// TwinCAT 3 PLC project PLC
// ProgramVersion: 3.1.4024.0
// libraries:
//   Tc2_Standard, * (Beckhoff Automation GmbH)
//   Tc2_System, * (Beckhoff Automation GmbH)
//   Tc3_Module, * (Beckhoff Automation GmbH)
// project tree:
//   / PlcTask.TcTTO
//   POUs/Alarm/ GVL_Alarm.TcGVL
//   POUs/EL3453/ FB_EL3453.TcPOU, stEL3453.TcDUT, stEL3453_ch.TcDUT, stEL3453_tot.TcDUT
//   POUs/Example/ GVL_HMI.TcGVL, GVL_IO.TcGVL, GVL_Safety.TcGVL, GVL_System.TcGVL, PRG_CircuitBreakerExample.TcPOU, PRG_ContactorExample.TcPOU, PRG_DisconnectorExample.TcPOU, PRG_Simulation.TcPOU
//   POUs/HVCP3/ GVL_HVCP3.TcGVL, PRG_HVCP3.TcPOU, PRG_HVCP3_14CB1.TcPOU, PRG_HVCP3_16CB1.TcPOU, PRG_HVCP3_18CB1.TcPOU, PRG_HVCP3_20CB1.TcPOU, PRG_HVCP3_22CB1.TcPOU, PRG_HVCP3_24CB1.TcPOU, PRG_HVCP3_26CB1.TcPOU, PRG_HVCP3_28CB1.TcPOU, PRG_HVCP3_30CB1.TcPOU, PRG_HVCP3_32CB1.TcPOU, PRG_HVCP3_34CB1.TcPOU, PRG_HVCP3_36CB1.TcPOU, PRG_HVCP3_38CB1.TcPOU, PRG_HVCP3_40CB1.TcPOU, PRG_HVCP3_42CB1.TcPOU, PRG_HVCP3_44CB1.TcPOU, PRG_HVCP3_46CB1.TcPOU, PRG_HVCP3_48CB1.TcPOU, PRG_HVCP3_50CB1.TcPOU, PRG_HVCP3_52CB1.TcPOU, PRG_HVCP3_54CB1.TcPOU, PRG_HVCP3_56CB1.TcPOU, PRG_HVCP3_10CB1.TcPOU, PRG_HVCP3_12CB1.TcPOU
//   POUs/HVCP5/ GVL_HVCP5.TcGVL, PRG_HVCP5.TcPOU, PRG_HVCP5_12CB1.TcPOU, PRG_HVCP5_14CB1.TcPOU, PRG_HVCP5_16CB1.TcPOU, PRG_HVCP5_18CB1.TcPOU, PRG_HVCP5_20CB1.TcPOU, PRG_HVCP5_22CB1.TcPOU, PRG_HVCP5_24CB1.TcPOU, PRG_HVCP5_26CB1.TcPOU, PRG_HVCP5_28CB1.TcPOU, PRG_HVCP5_30CB1.TcPOU, PRG_HVCP5_32CB1.TcPOU, PRG_HVCP5_34CB1.TcPOU, PRG_HVCP5_36CB1.TcPOU, PRG_HVCP5_38CB1.TcPOU, PRG_HVCP5_10CB1.TcPOU
//   POUs/LVCP1/ GVL_LVCP1.TcGVL, PRG_LVCP1_Colors.TcPOU, PRG_LVCP1_CompensationCalculate.TcPOU, PRG_LVCP1_Group1.TcPOU, PRG_LVCP1.TcPOU, PRG_LVCP1_Group2.TcPOU, PRG_LVCP1_Group3.TcPOU, PRG_LVCP1_Group4.TcPOU, PRG_LVCP1_Group5.TcPOU, PRG_LVCP1_Group10.TcPOU, PRG_LVCP1_Group9.TcPOU, PRG_LVCP1_Group8.TcPOU, PRG_LVCP1_Group7.TcPOU, PRG_LVCP1_Group6.TcPOU, PRG_LVCP1_MainDisconnector.TcPOU, PRG_LVCP1_PowerMeasurement.TcPOU
//   POUs/LVCP2/ GVL_LVCP2.TcGVL, PRG_LVCP2_Colors.TcPOU, PRG_LVCP2_PowerMeasurement.TcPOU, PRG_LVCP2.TcPOU, PRG_LVCP2_CompensationCalculate.TcPOU, PRG_LVCP2_Group10.TcPOU, PRG_LVCP2_Group1.TcPOU, PRG_LVCP2_Group2.TcPOU, PRG_LVCP2_Group3.TcPOU, PRG_LVCP2_Group4.TcPOU, PRG_LVCP2_Group5.TcPOU, PRG_LVCP2_Group6.TcPOU, PRG_LVCP2_Group7.TcPOU, PRG_LVCP2_Group8.TcPOU, PRG_LVCP2_Group9.TcPOU, PRG_LVCP2_MainDisconnector.TcPOU
//   POUs/LVCP5/ GVL_LVCP5.TcGVL, PRG_LVCP5_Colors.TcPOU, PRG_LVCP5_PowerMeasurement.TcPOU, PRG_LVCP5_CompensationCalculate.TcPOU, PRG_LVCP5_Group7.TcPOU, PRG_LVCP5_Group6.TcPOU, PRG_LVCP5_Group5.TcPOU, PRG_LVCP5_Group4.TcPOU, PRG_LVCP5_Group3.TcPOU, PRG_LVCP5_Group2.TcPOU, PRG_LVCP5_Group1.TcPOU, PRG_LVCP5.TcPOU, PRG_LVCP5_MainCircuitBreaker.TcPOU
//   POUs/ MAIN.TcPOU
//   _ES/11_Disconnector/Enum/ E_DisconnectorControlMode.TcTLEO, E_DisconnectorFault.TcTLEO, E_DisconnectorPosition.TcTLEO, E_DisconnectorStatus.TcTLEO
//   _ES/11_Disconnector/ FB_DisconnectorControl.TcPOU
//   _ES/11_Disconnector/Structure/ ST_DisconnectorCommand.TcDUT, ST_DisconnectorConfig.TcDUT, ST_DisconnectorHMI.TcDUT, ST_DisconnectorIO.TcDUT, ST_DisconnectorOperationRecord.TcDUT, ST_DisconnectorStatistics.TcDUT, ST_DisconnectorStatus.TcDUT
//   _ES/12_Contactor/Enum/ E_ContactorControlMode.TcTLEO, E_ContactorFault.TcTLEO, E_ContactorPosition.TcTLEO, E_ContactorStatus.TcTLEO
//   _ES/12_Contactor/ FB_ContactorControl.TcPOU
//   _ES/12_Contactor/Structure/ ST_ContactorCommand.TcDUT, ST_ContactorConfig.TcDUT, ST_ContactorHMI.TcDUT, ST_ContactorIO.TcDUT, ST_ContactorOperationRecord.TcDUT, ST_ContactorStatistics.TcDUT, ST_ContactorStatus.TcDUT
//   _ES/13_CircuitBreaker/Enum/ E_CircuitBreakerControlMode.TcTLEO, E_CircuitBreakerFault.TcTLEO, E_CircuitBreakerPosition.TcTLEO, E_CircuitBreakerStatus.TcTLEO
//   _ES/13_CircuitBreaker/ FB_CircuitBreaker.TcPOU
//   _ES/13_CircuitBreaker/Structure/ ST_CircuitBreakerCommand.TcDUT, ST_CircuitBreakerConfig.TcDUT, ST_CircuitBreakerHMI.TcDUT, ST_CircuitBreakerIO.TcDUT, ST_CircuitBreakerOperationRecord.TcDUT, ST_CircuitBreakerStatistics.TcDUT, ST_CircuitBreakerStatus.TcDUT
//   _ES/14_CompensationGroup/Enum/ E_CompensationError.TcTLEO
//   _ES/14_CompensationGroup/ FB_CompensationCalculator.TcPOU, GVL_CompensationGroup.TcGVL
//   _ES/14_CompensationGroup/Structure/ ST_CompensationConfigInfo.TcDUT, ST_CompensationDiagnostic.TcDUT, ST_CompensationGroup.TcDUT, ST_CompensationGroupDetails.TcDUT, ST_CompensationHMI.TcDUT, ST_CompensationSummary.TcDUT
//   _ES/xx_Line/Enum/ E_LineColors.TcDUT
//   _ES/xx_Line/Structure/ ST_CapacitorSchemaColorBase.TcDUT, ST_CapacitorSchemaColorWithContactor.TcDUT, ST_CapacitorSchemaColorWithDisconnector.TcDUT
// real-time tasks:
//   TASK PlcTask: cycle T#10ms, priority 20, ADS port 350
// I/O:
//   DEVICE Device 1 (EtherCAT) (disabled), AmsNetId 192.168.35.154.2.1
//     +EP6-11CP1 (EK1100) [EK1100 EtherCAT Coupler (2A E-Bus)]
//       +EP6-11DI1 (EL1809) [EL1809 16Ch. Dig. Input 24V, 3ms]
//       +EP6-11DI2 (EL1809) [EL1809 16Ch. Dig. Input 24V, 3ms]
//       +EP6-11DQ1 (EL2809-0015) [EL2809-0015 16Ch. Dig. Output 24V DC, 0.35A, not short-circuit proof]
//       +EP6-11SDI1 (EL1918) [EL1918, 8Ch. Safety Input 24V, TwinSAFE]
//         modules: Module 1 (FSOE), Module 2 (FSLOGIC)
//       +EP6-11SDQ1 (EL2904) [EL2904, 4 Ch. Safety Output 24V, 0.5A, TwinSAFE]
//         modules: Module 1 (FSOES), Module 2 (DO)
//       +EP6-11AI1 (EL3453) [EL3453 3Ch. Power Measuring]
//       Term 8 (EL9010) [EL9010 End Terminal]
//     +EP7-11CP1 (EK1100) [EK1100 EtherCAT Coupler (2A E-Bus)]
//       +EP7-11DI1 (EL1809) [EL1809 16Ch. Dig. Input 24V, 3ms]
//       +EP7-11DI2 (EL1809) [EL1809 16Ch. Dig. Input 24V, 3ms]
//       +EP7-11DQ1 (EL2809-0015) [EL2809-0015 16Ch. Dig. Output 24V DC, 0.35A, not short-circuit proof]
//       +EP7-11SDI1 (EL1918) [EL1918, 8Ch. Safety Input 24V, TwinSAFE]
//         modules: Module 1 (FSOE), Module 2 (FSLOGIC)
//       +EP7-11SDQ1 (EL2904) [EL2904, 4 Ch. Safety Output 24V, 0.5A, TwinSAFE]
//         modules: Module 1 (FSOES), Module 2 (DO)
//       +EP7-11AI1 (EL3453) [EL3453 3Ch. Power Measuring]
//       Term 16 (EL9010) [EL9010 End Terminal]
//     +EP8-11CP1 (EK1100) [EK1100 EtherCAT Coupler (2A E-Bus)]
//       +EP8-11DI1 (EL1809) [EL1809 16Ch. Dig. Input 24V, 3ms]
//       +EP8-11DI2 (EL1809) [EL1809 16Ch. Dig. Input 24V, 3ms]
//       +EP8-11DQ1 (EL2809-0015) [EL2809-0015 16Ch. Dig. Output 24V DC, 0.35A, not short-circuit proof]
//       +EP8-11SDI1 (EL1918) [EL1918, 8Ch. Safety Input 24V, TwinSAFE]
//         modules: Module 1 (FSOE), Module 2 (FSLOGIC)
//       +EP8-11SDQ1 (EL2904) [EL2904, 4 Ch. Safety Output 24V, 0.5A, TwinSAFE]
//         modules: Module 1 (FSOES), Module 2 (DO)
//       +EP8-11AI1 (EL3453) [EL3453 3Ch. Power Measuring]
//       Term 24 (EL9010) [EL9010 End Terminal]
//     +EP9-5CP5 (EK1100) [EK1100 EtherCAT Coupler (2A E-Bus)]
//       +EP9-5DI1 (EL1809) [EL1809 16Ch. Dig. Input 24V, 3ms]
//       +EP9-5DI2 (EL1809) [EL1809 16Ch. Dig. Input 24V, 3ms]
//       +EP9-5DI3 (EL1809) [EL1809 16Ch. Dig. Input 24V, 3ms]
//       +EP9-5DI4 (EL1809) [EL1809 16Ch. Dig. Input 24V, 3ms]
//       +EP9-5DI5 (EL1809) [EL1809 16Ch. Dig. Input 24V, 3ms]
//       +EP9-5DQ1 (EL2809) [EL2809 16Ch. Dig. Output 24V, 0.5A]
//       +EP9-5DQ2 (EL2809) [EL2809 16Ch. Dig. Output 24V, 0.5A]
//       +EP9-5DQ3 (EL2809) [EL2809 16Ch. Dig. Output 24V, 0.5A]
//       +EP9-6SDI1 (EL1918) [EL1918, 8Ch. Safety Input 24V, TwinSAFE]
//         modules: Module 1 (FSOE), Module 2 (FSLOGIC)
//       +EP9-6SDQ1 (EL2904) [EL2904, 4 Ch. Safety Output 24V, 0.5A, TwinSAFE]
//         modules: Module 1 (FSOES), Module 2 (DO)
//       +EP9-6AI1 (EL3453) [EL3453 3Ch. Power Measuring]
//     +EP10-5CP5 (EK1100) [EK1100 EtherCAT Coupler (2A E-Bus)]
//       +EP10-5DI1 (EL1809) [EL1809 16Ch. Dig. Input 24V, 3ms]
//       +EP10-5DI2 (EL1809) [EL1809 16Ch. Dig. Input 24V, 3ms]
//       +EP10-5DI3 (EL1809) [EL1809 16Ch. Dig. Input 24V, 3ms]
//       +EP10-5DI4 (EL1809) [EL1809 16Ch. Dig. Input 24V, 3ms]
//       +EP10-5DQ1 (EL2809) [EL2809 16Ch. Dig. Output 24V, 0.5A]
//       +EP10-5DQ2 (EL2809) [EL2809 16Ch. Dig. Output 24V, 0.5A]
//       +EP10-6SDI1 (EL1918) [EL1918, 8Ch. Safety Input 24V, TwinSAFE]
//         modules: Module 1 (FSOE), Module 2 (FSLOGIC)
//       +EP10-6SDQ1 (EL2904) [EL2904, 4 Ch. Safety Output 24V, 0.5A, TwinSAFE]
//         modules: Module 1 (FSOES), Module 2 (DO)
//       +EP10-6AI1 (EL3453) [EL3453 3Ch. Power Measuring]
// variable links:
//   PLC/PLC Instance <-> Device 1 (EtherCAT)/+EP10-5CP5 (EK1100)/+EP10-5DI1 (EL1809)
//     PlcTask Inputs/GVL_Alarm.EP10_3X2_24VDC_OK <-> Channel 1/Input
//     PlcTask Inputs/GVL_Alarm.EP10_UPS_24VDC_OK <-> Channel 2/Input
//     PlcTask Inputs/PRG_HVCP5_10CB1.stDisconnectorIO.bEarthSwitchOff <-> Channel 7/Input
//     PlcTask Inputs/PRG_HVCP5_10CB1.stDisconnectorIO.bEarthSwitchOn <-> Channel 6/Input
//     PlcTask Inputs/PRG_HVCP5_10CB1.stDisconnectorIO.bLimitOff <-> Channel 4/Input
//     PlcTask Inputs/PRG_HVCP5_12CB1.stDisconnectorIO.bLimitOff <-> Channel 9/Input
//     PlcTask Inputs/PRG_HVCP5_14CB1.stDisconnectorIO.bLimitOff <-> Channel 12/Input
//     PlcTask Inputs/PRG_HVCP5_16CB1.stDisconnectorIO.bLimitOff <-> Channel 15/Input
//     PlcTask Inputs/PRG_HVCP5_10CB1.stDisconnectorIO.bLimitOn <-> Channel 3/Input
//     PlcTask Inputs/PRG_HVCP5_12CB1.stDisconnectorIO.bLimitOn <-> Channel 8/Input
//     PlcTask Inputs/PRG_HVCP5_14CB1.stDisconnectorIO.bLimitOn <-> Channel 11/Input
//     PlcTask Inputs/PRG_HVCP5_16CB1.stDisconnectorIO.bLimitOn <-> Channel 14/Input
//     PlcTask Inputs/PRG_HVCP5_10CB1.stDisconnectorIO.bPLCControl <-> Channel 5/Input
//     PlcTask Inputs/PRG_HVCP5_12CB1.stDisconnectorIO.bPLCControl <-> Channel 10/Input
//     PlcTask Inputs/PRG_HVCP5_14CB1.stDisconnectorIO.bPLCControl <-> Channel 13/Input
//     PlcTask Inputs/PRG_HVCP5_16CB1.stDisconnectorIO.bPLCControl <-> Channel 16/Input
//   PLC/PLC Instance <-> Device 1 (EtherCAT)/+EP10-5CP5 (EK1100)/+EP10-5DI2 (EL1809)
//     PlcTask Inputs/PRG_HVCP5_{18..26 step 2}CB1.stDisconnectorIO.bLimitOff <-> Channel {2..14 step 3}/Input  (5 links)
//     PlcTask Inputs/PRG_HVCP5_{18..28 step 2}CB1.stDisconnectorIO.bLimitOn <-> Channel {1..16 step 3}/Input  (6 links)
//     PlcTask Inputs/PRG_HVCP5_{18..26 step 2}CB1.stDisconnectorIO.bPLCControl <-> Channel {3..15 step 3}/Input  (5 links)
//   PLC/PLC Instance <-> Device 1 (EtherCAT)/+EP10-5CP5 (EK1100)/+EP10-5DI3 (EL1809)
//     PlcTask Inputs/PRG_HVCP5_{28..38 step 2}CB1.stDisconnectorIO.bLimitOff <-> Channel {1..16 step 3}/Input  (6 links)
//     PlcTask Inputs/PRG_HVCP5_{28..36 step 2}CB1.stDisconnectorIO.bPLCControl <-> Channel {2..14 step 3}/Input  (5 links)
//     PlcTask Inputs/PRG_HVCP5_{30..38 step 2}CB1.stDisconnectorIO.bLimitOn <-> Channel {3..15 step 3}/Input  (5 links)
//   PLC/PLC Instance <-> Device 1 (EtherCAT)/+EP10-5CP5 (EK1100)/+EP10-5DI4 (EL1809)
//     PlcTask Inputs/PRG_HVCP5_38CB1.stDisconnectorIO.bPLCControl <-> Channel 1/Input
//   PLC/PLC Instance <-> Device 1 (EtherCAT)/+EP10-5CP5 (EK1100)/+EP10-5DQ1 (EL2809)
//     PlcTask Outputs/PRG_HVCP5_{10..24 step 2}CB1.stDisconnectorIO.bContactorOff_Out <-> Channel {2..16 step 2}/Output  (8 links)
//     PlcTask Outputs/PRG_HVCP5_{10..24 step 2}CB1.stDisconnectorIO.bContactorOn_Out <-> Channel {1..15 step 2}/Output  (8 links)
//   PLC/PLC Instance <-> Device 1 (EtherCAT)/+EP10-5CP5 (EK1100)/+EP10-5DQ2 (EL2809)
//     PlcTask Outputs/PRG_HVCP5_{26..38 step 2}CB1.stDisconnectorIO.bContactorOff_Out <-> Channel {2..14 step 2}/Output  (7 links)
//     PlcTask Outputs/PRG_HVCP5_{26..38 step 2}CB1.stDisconnectorIO.bContactorOn_Out <-> Channel {1..13 step 2}/Output  (7 links)
//   PLC/PLC Instance <-> Device 1 (EtherCAT)/+EP6-11CP1 (EK1100)/+EP6-11AI1 (EL3453)
//     PlcTask Inputs/PRG_LVCP1_PowerMeasurement.fbEL3453.EL3453.MDP5001_341_Input/MDP5001_341_L1_Basic_Current <-> L1 Basic/Current
//     PlcTask Inputs/PRG_LVCP1_PowerMeasurement.fbEL3453.EL3453.MDP5001_341_Input/MDP5001_341_L2_Basic_Current <-> L2 Basic/Current
//     PlcTask Inputs/PRG_LVCP1_PowerMeasurement.fbEL3453.EL3453.MDP5001_341_Input/MDP5001_341_L3_Basic_Current <-> L3 Basic/Current
//     PlcTask Inputs/PRG_LVCP1_PowerMeasurement.fbEL3453.EL3453.MDP5001_341_Input/MDP5001_341_L1_Basic_Voltage <-> L1 Basic/Voltage
//     PlcTask Inputs/PRG_LVCP1_PowerMeasurement.fbEL3453.EL3453.MDP5001_341_Input/MDP5001_341_L2_Basic_Voltage <-> L2 Basic/Voltage
//     PlcTask Inputs/PRG_LVCP1_PowerMeasurement.fbEL3453.EL3453.MDP5001_341_Input/MDP5001_341_L3_Basic_Voltage <-> L3 Basic/Voltage
//     PlcTask Inputs/PRG_LVCP1_PowerMeasurement.fbEL3453.EL3453.MDP5001_341_Input/MDP5001_341_L1_Power_Active_Power <-> L1 Power/Active Power
//     PlcTask Inputs/PRG_LVCP1_PowerMeasurement.fbEL3453.EL3453.MDP5001_341_Input/MDP5001_341_L2_Power_Active_Power <-> L2 Power/Active Power
//     PlcTask Inputs/PRG_LVCP1_PowerMeasurement.fbEL3453.EL3453.MDP5001_341_Input/MDP5001_341_L3_Power_Active_Power <-> L3 Power/Active Power
//     PlcTask Inputs/PRG_LVCP1_PowerMeasurement.fbEL3453.EL3453.MDP5001_341_Input/MDP5001_341_L1_Power_Apparent_Power <-> L1 Power/Apparent Power
//     PlcTask Inputs/PRG_LVCP1_PowerMeasurement.fbEL3453.EL3453.MDP5001_341_Input/MDP5001_341_L2_Power_Apparent_Power <-> L2 Power/Apparent Power
//     PlcTask Inputs/PRG_LVCP1_PowerMeasurement.fbEL3453.EL3453.MDP5001_341_Input/MDP5001_341_L3_Power_Apparent_Power <-> L3 Power/Apparent Power
//     PlcTask Inputs/PRG_LVCP1_PowerMeasurement.fbEL3453.EL3453.MDP5001_341_Input/MDP5001_341_L1_Power_Power_Factor <-> L1 Power/Power Factor
//     PlcTask Inputs/PRG_LVCP1_PowerMeasurement.fbEL3453.EL3453.MDP5001_341_Input/MDP5001_341_L2_Power_Power_Factor <-> L2 Power/Power Factor
//     PlcTask Inputs/PRG_LVCP1_PowerMeasurement.fbEL3453.EL3453.MDP5001_341_Input/MDP5001_341_L3_Power_Power_Factor <-> L3 Power/Power Factor
//     PlcTask Inputs/PRG_LVCP1_PowerMeasurement.fbEL3453.EL3453.MDP5001_341_Input/MDP5001_341_L1_Power_Reactive_Power <-> L1 Power/Reactive Power
//     PlcTask Inputs/PRG_LVCP1_PowerMeasurement.fbEL3453.EL3453.MDP5001_341_Input/MDP5001_341_L2_Power_Reactive_Power <-> L2 Power/Reactive Power
//     PlcTask Inputs/PRG_LVCP1_PowerMeasurement.fbEL3453.EL3453.MDP5001_341_Input/MDP5001_341_L3_Power_Reactive_Power <-> L3 Power/Reactive Power
//     PlcTask Inputs/PRG_LVCP1_PowerMeasurement.fbEL3453.EL3453.MDP5001_341_Input/MDP5001_341_L1_Status_Current_Guard_Error <-> L1 Status/Current Guard Error
//     PlcTask Inputs/PRG_LVCP1_PowerMeasurement.fbEL3453.EL3453.MDP5001_341_Input/MDP5001_341_L2_Status_Current_Guard_Error <-> L2 Status/Current Guard Error
//     PlcTask Inputs/PRG_LVCP1_PowerMeasurement.fbEL3453.EL3453.MDP5001_341_Input/MDP5001_341_L3_Status_Current_Guard_Error <-> L3 Status/Current Guard Error
//     PlcTask Inputs/PRG_LVCP1_PowerMeasurement.fbEL3453.EL3453.MDP5001_341_Input/MDP5001_341_L1_Status_Current_Guard_Warning <-> L1 Status/Current Guard Warning
//     PlcTask Inputs/PRG_LVCP1_PowerMeasurement.fbEL3453.EL3453.MDP5001_341_Input/MDP5001_341_L2_Status_Current_Guard_Warning <-> L2 Status/Current Guard Warning
//     PlcTask Inputs/PRG_LVCP1_PowerMeasurement.fbEL3453.EL3453.MDP5001_341_Input/MDP5001_341_L3_Status_Current_Guard_Warning <-> L3 Status/Current Guard Warning
//     PlcTask Inputs/PRG_LVCP1_PowerMeasurement.fbEL3453.EL3453.MDP5001_341_Input/MDP5001_341_L1_Status_Inaccurate_Current <-> L1 Status/Inaccurate Current
//     PlcTask Inputs/PRG_LVCP1_PowerMeasurement.fbEL3453.EL3453.MDP5001_341_Input/MDP5001_341_L2_Status_Inaccurate_Current <-> L2 Status/Inaccurate Current
//     PlcTask Inputs/PRG_LVCP1_PowerMeasurement.fbEL3453.EL3453.MDP5001_341_Input/MDP5001_341_L3_Status_Inaccurate_Current <-> L3 Status/Inaccurate Current
//     PlcTask Inputs/PRG_LVCP1_PowerMeasurement.fbEL3453.EL3453.MDP5001_341_Input/MDP5001_341_L1_Status_Inaccurate_Voltage <-> L1 Status/Inaccurate Voltage
//     PlcTask Inputs/PRG_LVCP1_PowerMeasurement.fbEL3453.EL3453.MDP5001_341_Input/MDP5001_341_L2_Status_Inaccurate_Voltage <-> L2 Status/Inaccurate Voltage
//     PlcTask Inputs/PRG_LVCP1_PowerMeasurement.fbEL3453.EL3453.MDP5001_341_Input/MDP5001_341_L3_Status_Inaccurate_Voltage <-> L3 Status/Inaccurate Voltage
//     PlcTask Inputs/PRG_LVCP1_PowerMeasurement.fbEL3453.EL3453.MDP5001_341_Input/MDP5001_341_L1_Status_Overcurrent <-> L1 Status/Overcurrent
//     PlcTask Inputs/PRG_LVCP1_PowerMeasurement.fbEL3453.EL3453.MDP5001_341_Input/MDP5001_341_L2_Status_Overcurrent <-> L2 Status/Overcurrent
//     PlcTask Inputs/PRG_LVCP1_PowerMeasurement.fbEL3453.EL3453.MDP5001_341_Input/MDP5001_341_L3_Status_Overcurrent <-> L3 Status/Overcurrent
//     PlcTask Inputs/PRG_LVCP1_PowerMeasurement.fbEL3453.EL3453.MDP5001_341_Input/MDP5001_341_L1_Status_Overvoltage <-> L1 Status/Overvoltage
//     PlcTask Inputs/PRG_LVCP1_PowerMeasurement.fbEL3453.EL3453.MDP5001_341_Input/MDP5001_341_L2_Status_Overvoltage <-> L2 Status/Overvoltage
//     PlcTask Inputs/PRG_LVCP1_PowerMeasurement.fbEL3453.EL3453.MDP5001_341_Input/MDP5001_341_L3_Status_Overvoltage <-> L3 Status/Overvoltage
//     PlcTask Inputs/PRG_LVCP1_PowerMeasurement.fbEL3453.EL3453.MDP5001_341_Input/MDP5001_341_L1_Status_TxPDO_Toggle <-> L1 Status/TxPDO Toggle
//     PlcTask Inputs/PRG_LVCP1_PowerMeasurement.fbEL3453.EL3453.MDP5001_341_Input/MDP5001_341_L2_Status_TxPDO_Toggle <-> L2 Status/TxPDO Toggle
//     PlcTask Inputs/PRG_LVCP1_PowerMeasurement.fbEL3453.EL3453.MDP5001_341_Input/MDP5001_341_L3_Status_TxPDO_Toggle <-> L3 Status/TxPDO Toggle
//     PlcTask Inputs/PRG_LVCP1_PowerMeasurement.fbEL3453.EL3453.MDP5001_341_Input/MDP5001_341_L1_Status_Voltage_Guard_Error <-> L1 Status/Voltage Guard Error
//     PlcTask Inputs/PRG_LVCP1_PowerMeasurement.fbEL3453.EL3453.MDP5001_341_Input/MDP5001_341_L2_Status_Voltage_Guard_Error <-> L2 Status/Voltage Guard Error
//     PlcTask Inputs/PRG_LVCP1_PowerMeasurement.fbEL3453.EL3453.MDP5001_341_Input/MDP5001_341_L3_Status_Voltage_Guard_Error <-> L3 Status/Voltage Guard Error
//     PlcTask Inputs/PRG_LVCP1_PowerMeasurement.fbEL3453.EL3453.MDP5001_341_Input/MDP5001_341_L1_Status_Voltage_Guard_Warning <-> L1 Status/Voltage Guard Warning
//     PlcTask Inputs/PRG_LVCP1_PowerMeasurement.fbEL3453.EL3453.MDP5001_341_Input/MDP5001_341_L2_Status_Voltage_Guard_Warning <-> L2 Status/Voltage Guard Warning
//     PlcTask Inputs/PRG_LVCP1_PowerMeasurement.fbEL3453.EL3453.MDP5001_341_Input/MDP5001_341_L3_Status_Voltage_Guard_Warning <-> L3 Status/Voltage Guard Warning
//     PlcTask Inputs/PRG_LVCP1_PowerMeasurement.fbEL3453.EL3453.MDP5001_341_Input/MDP5001_341_L1_Status_Voltage_Sign_Bit <-> L1 Status/Voltage Sign Bit
//     PlcTask Inputs/PRG_LVCP1_PowerMeasurement.fbEL3453.EL3453.MDP5001_341_Input/MDP5001_341_L2_Status_Voltage_Sign_Bit <-> L2 Status/Voltage Sign Bit
//     PlcTask Inputs/PRG_LVCP1_PowerMeasurement.fbEL3453.EL3453.MDP5001_341_Input/MDP5001_341_L3_Status_Voltage_Sign_Bit <-> L3 Status/Voltage Sign Bit
//     PlcTask Inputs/PRG_LVCP1_PowerMeasurement.fbEL3453.EL3453.MDP5001_341_Input/MDP5001_341_Total_Basic_Calculated_Error_Current <-> Total Basic/Calculated Error Current
//     PlcTask Inputs/PRG_LVCP1_PowerMeasurement.fbEL3453.EL3453.MDP5001_341_Input/MDP5001_341_Total_Basic_Frequency <-> Total Basic/Frequency
//     PlcTask Inputs/PRG_LVCP1_PowerMeasurement.fbEL3453.EL3453.MDP5001_341_Input/MDP5001_341_Total_Basic_Neutral_Line_Current <-> Total Basic/Neutral Line Current
//     PlcTask Inputs/PRG_LVCP1_PowerMeasurement.fbEL3453.EL3453.MDP5001_341_Input/MDP5001_341_Total_Basic_Power_Factor <-> Total Basic/Power Factor
//     PlcTask Inputs/PRG_LVCP1_PowerMeasurement.fbEL3453.EL3453.MDP5001_341_Input/MDP5001_341_Total_Basic_ROCOF <-> Total Basic/ROCOF
//     PlcTask Inputs/PRG_LVCP1_PowerMeasurement.fbEL3453.EL3453.MDP5001_341_Input/MDP5001_341_Total_Status_Active_Power_Guard_Error <-> Total Status/Active Power Guard Error
//     PlcTask Inputs/PRG_LVCP1_PowerMeasurement.fbEL3453.EL3453.MDP5001_341_Input/MDP5001_341_Total_Status_Active_Power_Guard_Warning <-> Total Status/Active Power Guard Warning
//     PlcTask Inputs/PRG_LVCP1_PowerMeasurement.fbEL3453.EL3453.MDP5001_341_Input/MDP5001_341_Total_Status_Apparent_Power_Guard_Error <-> Total Status/Apparent Power Guard Error
//     PlcTask Inputs/PRG_LVCP1_PowerMeasurement.fbEL3453.EL3453.MDP5001_341_Input/MDP5001_341_Total_Status_Apparent_Power_Guard_Warning <-> Total Status/Apparent Power Guard Warning
//     PlcTask Inputs/PRG_LVCP1_PowerMeasurement.fbEL3453.EL3453.MDP5001_341_Input/MDP5001_341_Total_Status_Frequency_Guard_Error <-> Total Status/Frequency Guard Error
//     PlcTask Inputs/PRG_LVCP1_PowerMeasurement.fbEL3453.EL3453.MDP5001_341_Input/MDP5001_341_Total_Status_Frequency_Guard_Warning <-> Total Status/Frequency Guard Warning
//     PlcTask Inputs/PRG_LVCP1_PowerMeasurement.fbEL3453.EL3453.MDP5001_341_Input/MDP5001_341_Total_Status_Grid_Direction <-> Total Status/Grid Direction
//     PlcTask Inputs/PRG_LVCP1_PowerMeasurement.fbEL3453.EL3453.MDP5001_341_Input/MDP5001_341_Total_Status_Neutral_Current_Guard_Error <-> Total Status/Neutral Current Guard Error
//     PlcTask Inputs/PRG_LVCP1_PowerMeasurement.fbEL3453.EL3453.MDP5001_341_Input/MDP5001_341_Total_Status_Neutral_Current_Guard_Warning <-> Total Status/Neutral Current Guard Warning
//     PlcTask Inputs/PRG_LVCP1_PowerMeasurement.fbEL3453.EL3453.MDP5001_341_Input/MDP5001_341_Total_Status_Power_Quality_Factor <-> Total Status/Power Quality Factor
//     PlcTask Inputs/PRG_LVCP1_PowerMeasurement.fbEL3453.EL3453.MDP5001_341_Input/MDP5001_341_Total_Status_Power_Quality_Guard_Error <-> Total Status/Power Quality Guard Error
//     PlcTask Inputs/PRG_LVCP1_PowerMeasurement.fbEL3453.EL3453.MDP5001_341_Input/MDP5001_341_Total_Status_Power_Quality_Guard_Warning <-> Total Status/Power Quality Guard Warning
//     PlcTask Inputs/PRG_LVCP1_PowerMeasurement.fbEL3453.EL3453.MDP5001_341_Input/MDP5001_341_Total_Status_System_State <-> Total Status/System State
//     PlcTask Inputs/PRG_LVCP1_PowerMeasurement.fbEL3453.EL3453.MDP5001_341_Input/MDP5001_341_Total_Status_TxPDO_State <-> Total Status/TxPDO State
//     PlcTask Inputs/PRG_LVCP1_PowerMeasurement.fbEL3453.EL3453.MDP5001_341_Input/MDP5001_341_Total_Status_TxPDO_Toggle <-> Total Status/TxPDO Toggle
//     PlcTask Inputs/PRG_LVCP1_PowerMeasurement.fbEL3453.EL3453.MDP5001_341_Input/MDP5001_341_Total_Variant_Value_In_Index_1_REAL <-> Total Variant Value In/Index 1 REAL
//     PlcTask Inputs/PRG_LVCP1_PowerMeasurement.fbEL3453.EL3453.MDP5001_341_Input/MDP5001_341_Total_Variant_Value_In_Index_2_REAL <-> Total Variant Value In/Index 2 REAL
//     PlcTask Inputs/PRG_LVCP1_PowerMeasurement.fbEL3453.EL3453.MDP5001_341_Input/MDP5001_341_Total_Variant_Value_In_Index_3_REAL <-> Total Variant Value In/Index 3 REAL
//     PlcTask Inputs/PRG_LVCP1_PowerMeasurement.fbEL3453.EL3453.MDP5001_341_Input/MDP5001_341_Total_Variant_Value_In_Index_4_ULINT <-> Total Variant Value In/Index 4 ULINT
//     PlcTask Inputs/PRG_LVCP1_PowerMeasurement.fbEL3453.EL3453.MDP5001_341_Input/MDP5001_341_Total_Variant_Value_In_TxPDO_Toggle <-> Total Variant Value In/TxPDO Toggle
//     PlcTask Inputs/PRG_LVCP1_PowerMeasurement.fbEL3453.EL3453.MDP5001_341_Input/MDP5001_341_Total_Variant_Value_In_Value_1_REAL <-> Total Variant Value In/Value 1 REAL
//     PlcTask Inputs/PRG_LVCP1_PowerMeasurement.fbEL3453.EL3453.MDP5001_341_Input/MDP5001_341_Total_Variant_Value_In_Value_2_REAL <-> Total Variant Value In/Value 2 REAL
//     PlcTask Inputs/PRG_LVCP1_PowerMeasurement.fbEL3453.EL3453.MDP5001_341_Input/MDP5001_341_Total_Variant_Value_In_Value_3_REAL <-> Total Variant Value In/Value 3 REAL
//     PlcTask Inputs/PRG_LVCP1_PowerMeasurement.fbEL3453.EL3453.MDP5001_341_Input/MDP5001_341_Total_Variant_Value_In_Value_4_ULINT <-> Total Variant Value In/Value 4 ULINT
//     PlcTask Outputs/PRG_LVCP1_PowerMeasurement.fbEL3453.EL3453.MDP5001_341_Output/MDP5001_341_Total_Variant_Value_Out_Index_1_REAL <-> Total Variant Value Out/Index 1 REAL
//     PlcTask Outputs/PRG_LVCP1_PowerMeasurement.fbEL3453.EL3453.MDP5001_341_Output/MDP5001_341_Total_Variant_Value_Out_Index_2_REAL <-> Total Variant Value Out/Index 2 REAL
//     PlcTask Outputs/PRG_LVCP1_PowerMeasurement.fbEL3453.EL3453.MDP5001_341_Output/MDP5001_341_Total_Variant_Value_Out_Index_3_REAL <-> Total Variant Value Out/Index 3 REAL
//     PlcTask Outputs/PRG_LVCP1_PowerMeasurement.fbEL3453.EL3453.MDP5001_341_Output/MDP5001_341_Total_Variant_Value_Out_Index_4_ULINT <-> Total Variant Value Out/Index 4 ULINT
//   PLC/PLC Instance <-> Device 1 (EtherCAT)/+EP6-11CP1 (EK1100)/+EP6-11DI1 (EL1809)
//     PlcTask Inputs/GVL_Alarm.EP6_3X2_24VDC_OK <-> Channel 1/Input
//     PlcTask Inputs/GVL_Alarm.EP6_UPS_24VDC_OK <-> Channel 2/Input
//     PlcTask Inputs/PRG_LVCP1_Group{1..6}.stContactor_IO.bFeedback <-> Channel {6..16 step 2}/Input  (6 links)
//     PlcTask Inputs/PRG_LVCP1_Group{1..5}.stContactor_IO.bPLCControl <-> Channel {7..15 step 2}/Input  (5 links)
//     PlcTask Inputs/PRG_LVCP1_MainDisconnector.stDisconnectorIO.bContactorOff_FB <-> Channel 4/Input
//     PlcTask Inputs/PRG_LVCP1_MainDisconnector.stDisconnectorIO.bContactorOn_FB <-> Channel 3/Input
//     PlcTask Inputs/PRG_LVCP1_MainDisconnector.stDisconnectorIO.bPLCControl <-> Channel 5/Input
//   PLC/PLC Instance <-> Device 1 (EtherCAT)/+EP6-11CP1 (EK1100)/+EP6-11DI2 (EL1809)
//     PlcTask Inputs/PRG_LVCP1_Group{7..10}.stContactor_IO.bFeedback <-> Channel {2..8 step 2}/Input  (4 links)
//     PlcTask Inputs/PRG_LVCP1_Group{6..10}.stContactor_IO.bPLCControl <-> Channel {1..9 step 2}/Input  (5 links)
//   PLC/PLC Instance <-> Device 1 (EtherCAT)/+EP6-11CP1 (EK1100)/+EP6-11DQ1 (EL2809-0015)
//     PlcTask Outputs/PRG_LVCP1_Group{1..10}.stContactor_IO.bOutput <-> Channel {3..12}/Output  (10 links)
//     PlcTask Outputs/PRG_LVCP1_MainDisconnector.stDisconnectorIO.bContactorOff_Out <-> Channel 2/Output
//     PlcTask Outputs/PRG_LVCP1_MainDisconnector.stDisconnectorIO.bContactorOn_Out <-> Channel 1/Output
//   PLC/PLC Instance <-> Device 1 (EtherCAT)/+EP7-11CP1 (EK1100)/+EP7-11AI1 (EL3453)
//     PlcTask Inputs/PRG_LVCP2_PowerMeasurement.fbEL3453.EL3453.MDP5001_341_Input/MDP5001_341_L1_Basic_Current <-> L1 Basic/Current
//     PlcTask Inputs/PRG_LVCP2_PowerMeasurement.fbEL3453.EL3453.MDP5001_341_Input/MDP5001_341_L2_Basic_Current <-> L2 Basic/Current
//     PlcTask Inputs/PRG_LVCP2_PowerMeasurement.fbEL3453.EL3453.MDP5001_341_Input/MDP5001_341_L3_Basic_Current <-> L3 Basic/Current
//     PlcTask Inputs/PRG_LVCP2_PowerMeasurement.fbEL3453.EL3453.MDP5001_341_Input/MDP5001_341_L1_Basic_Voltage <-> L1 Basic/Voltage
//     PlcTask Inputs/PRG_LVCP2_PowerMeasurement.fbEL3453.EL3453.MDP5001_341_Input/MDP5001_341_L2_Basic_Voltage <-> L2 Basic/Voltage
//     PlcTask Inputs/PRG_LVCP2_PowerMeasurement.fbEL3453.EL3453.MDP5001_341_Input/MDP5001_341_L3_Basic_Voltage <-> L3 Basic/Voltage
//     PlcTask Inputs/PRG_LVCP2_PowerMeasurement.fbEL3453.EL3453.MDP5001_341_Input/MDP5001_341_L1_Power_Active_Power <-> L1 Power/Active Power
//     PlcTask Inputs/PRG_LVCP2_PowerMeasurement.fbEL3453.EL3453.MDP5001_341_Input/MDP5001_341_L2_Power_Active_Power <-> L2 Power/Active Power
//     PlcTask Inputs/PRG_LVCP2_PowerMeasurement.fbEL3453.EL3453.MDP5001_341_Input/MDP5001_341_L3_Power_Active_Power <-> L3 Power/Active Power
//     PlcTask Inputs/PRG_LVCP2_PowerMeasurement.fbEL3453.EL3453.MDP5001_341_Input/MDP5001_341_L1_Power_Apparent_Power <-> L1 Power/Apparent Power
//     PlcTask Inputs/PRG_LVCP2_PowerMeasurement.fbEL3453.EL3453.MDP5001_341_Input/MDP5001_341_L2_Power_Apparent_Power <-> L2 Power/Apparent Power
//     PlcTask Inputs/PRG_LVCP2_PowerMeasurement.fbEL3453.EL3453.MDP5001_341_Input/MDP5001_341_L3_Power_Apparent_Power <-> L3 Power/Apparent Power
//     PlcTask Inputs/PRG_LVCP2_PowerMeasurement.fbEL3453.EL3453.MDP5001_341_Input/MDP5001_341_L1_Power_Power_Factor <-> L1 Power/Power Factor
//     PlcTask Inputs/PRG_LVCP2_PowerMeasurement.fbEL3453.EL3453.MDP5001_341_Input/MDP5001_341_L2_Power_Power_Factor <-> L2 Power/Power Factor
//     PlcTask Inputs/PRG_LVCP2_PowerMeasurement.fbEL3453.EL3453.MDP5001_341_Input/MDP5001_341_L3_Power_Power_Factor <-> L3 Power/Power Factor
//     PlcTask Inputs/PRG_LVCP2_PowerMeasurement.fbEL3453.EL3453.MDP5001_341_Input/MDP5001_341_L1_Power_Reactive_Power <-> L1 Power/Reactive Power
//     PlcTask Inputs/PRG_LVCP2_PowerMeasurement.fbEL3453.EL3453.MDP5001_341_Input/MDP5001_341_L2_Power_Reactive_Power <-> L2 Power/Reactive Power
//     PlcTask Inputs/PRG_LVCP2_PowerMeasurement.fbEL3453.EL3453.MDP5001_341_Input/MDP5001_341_L3_Power_Reactive_Power <-> L3 Power/Reactive Power
//     PlcTask Inputs/PRG_LVCP2_PowerMeasurement.fbEL3453.EL3453.MDP5001_341_Input/MDP5001_341_L1_Status_Current_Guard_Error <-> L1 Status/Current Guard Error
//     PlcTask Inputs/PRG_LVCP2_PowerMeasurement.fbEL3453.EL3453.MDP5001_341_Input/MDP5001_341_L2_Status_Current_Guard_Error <-> L2 Status/Current Guard Error
//     PlcTask Inputs/PRG_LVCP2_PowerMeasurement.fbEL3453.EL3453.MDP5001_341_Input/MDP5001_341_L3_Status_Current_Guard_Error <-> L3 Status/Current Guard Error
//     PlcTask Inputs/PRG_LVCP2_PowerMeasurement.fbEL3453.EL3453.MDP5001_341_Input/MDP5001_341_L1_Status_Current_Guard_Warning <-> L1 Status/Current Guard Warning
//     PlcTask Inputs/PRG_LVCP2_PowerMeasurement.fbEL3453.EL3453.MDP5001_341_Input/MDP5001_341_L2_Status_Current_Guard_Warning <-> L2 Status/Current Guard Warning
//     PlcTask Inputs/PRG_LVCP2_PowerMeasurement.fbEL3453.EL3453.MDP5001_341_Input/MDP5001_341_L3_Status_Current_Guard_Warning <-> L3 Status/Current Guard Warning
//     PlcTask Inputs/PRG_LVCP2_PowerMeasurement.fbEL3453.EL3453.MDP5001_341_Input/MDP5001_341_L1_Status_Inaccurate_Current <-> L1 Status/Inaccurate Current
//     PlcTask Inputs/PRG_LVCP2_PowerMeasurement.fbEL3453.EL3453.MDP5001_341_Input/MDP5001_341_L2_Status_Inaccurate_Current <-> L2 Status/Inaccurate Current
//     PlcTask Inputs/PRG_LVCP2_PowerMeasurement.fbEL3453.EL3453.MDP5001_341_Input/MDP5001_341_L3_Status_Inaccurate_Current <-> L3 Status/Inaccurate Current
//     PlcTask Inputs/PRG_LVCP2_PowerMeasurement.fbEL3453.EL3453.MDP5001_341_Input/MDP5001_341_L1_Status_Inaccurate_Voltage <-> L1 Status/Inaccurate Voltage
//     PlcTask Inputs/PRG_LVCP2_PowerMeasurement.fbEL3453.EL3453.MDP5001_341_Input/MDP5001_341_L2_Status_Inaccurate_Voltage <-> L2 Status/Inaccurate Voltage
//     PlcTask Inputs/PRG_LVCP2_PowerMeasurement.fbEL3453.EL3453.MDP5001_341_Input/MDP5001_341_L3_Status_Inaccurate_Voltage <-> L3 Status/Inaccurate Voltage
//     PlcTask Inputs/PRG_LVCP2_PowerMeasurement.fbEL3453.EL3453.MDP5001_341_Input/MDP5001_341_L1_Status_Overcurrent <-> L1 Status/Overcurrent
//     PlcTask Inputs/PRG_LVCP2_PowerMeasurement.fbEL3453.EL3453.MDP5001_341_Input/MDP5001_341_L2_Status_Overcurrent <-> L2 Status/Overcurrent
//     PlcTask Inputs/PRG_LVCP2_PowerMeasurement.fbEL3453.EL3453.MDP5001_341_Input/MDP5001_341_L3_Status_Overcurrent <-> L3 Status/Overcurrent
//     PlcTask Inputs/PRG_LVCP2_PowerMeasurement.fbEL3453.EL3453.MDP5001_341_Input/MDP5001_341_L1_Status_Overvoltage <-> L1 Status/Overvoltage
//     PlcTask Inputs/PRG_LVCP2_PowerMeasurement.fbEL3453.EL3453.MDP5001_341_Input/MDP5001_341_L2_Status_Overvoltage <-> L2 Status/Overvoltage
//     PlcTask Inputs/PRG_LVCP2_PowerMeasurement.fbEL3453.EL3453.MDP5001_341_Input/MDP5001_341_L3_Status_Overvoltage <-> L3 Status/Overvoltage
//     PlcTask Inputs/PRG_LVCP2_PowerMeasurement.fbEL3453.EL3453.MDP5001_341_Input/MDP5001_341_L1_Status_TxPDO_Toggle <-> L1 Status/TxPDO Toggle
//     PlcTask Inputs/PRG_LVCP2_PowerMeasurement.fbEL3453.EL3453.MDP5001_341_Input/MDP5001_341_L2_Status_TxPDO_Toggle <-> L2 Status/TxPDO Toggle
//     PlcTask Inputs/PRG_LVCP2_PowerMeasurement.fbEL3453.EL3453.MDP5001_341_Input/MDP5001_341_L3_Status_TxPDO_Toggle <-> L3 Status/TxPDO Toggle
//     PlcTask Inputs/PRG_LVCP2_PowerMeasurement.fbEL3453.EL3453.MDP5001_341_Input/MDP5001_341_L1_Status_Voltage_Guard_Error <-> L1 Status/Voltage Guard Error
//     PlcTask Inputs/PRG_LVCP2_PowerMeasurement.fbEL3453.EL3453.MDP5001_341_Input/MDP5001_341_L2_Status_Voltage_Guard_Error <-> L2 Status/Voltage Guard Error
//     PlcTask Inputs/PRG_LVCP2_PowerMeasurement.fbEL3453.EL3453.MDP5001_341_Input/MDP5001_341_L3_Status_Voltage_Guard_Error <-> L3 Status/Voltage Guard Error
//     PlcTask Inputs/PRG_LVCP2_PowerMeasurement.fbEL3453.EL3453.MDP5001_341_Input/MDP5001_341_L1_Status_Voltage_Guard_Warning <-> L1 Status/Voltage Guard Warning
//     PlcTask Inputs/PRG_LVCP2_PowerMeasurement.fbEL3453.EL3453.MDP5001_341_Input/MDP5001_341_L2_Status_Voltage_Guard_Warning <-> L2 Status/Voltage Guard Warning
//     PlcTask Inputs/PRG_LVCP2_PowerMeasurement.fbEL3453.EL3453.MDP5001_341_Input/MDP5001_341_L3_Status_Voltage_Guard_Warning <-> L3 Status/Voltage Guard Warning
//     PlcTask Inputs/PRG_LVCP2_PowerMeasurement.fbEL3453.EL3453.MDP5001_341_Input/MDP5001_341_L1_Status_Voltage_Sign_Bit <-> L1 Status/Voltage Sign Bit
//     PlcTask Inputs/PRG_LVCP2_PowerMeasurement.fbEL3453.EL3453.MDP5001_341_Input/MDP5001_341_L2_Status_Voltage_Sign_Bit <-> L2 Status/Voltage Sign Bit
//     PlcTask Inputs/PRG_LVCP2_PowerMeasurement.fbEL3453.EL3453.MDP5001_341_Input/MDP5001_341_L3_Status_Voltage_Sign_Bit <-> L3 Status/Voltage Sign Bit
//     PlcTask Inputs/PRG_LVCP2_PowerMeasurement.fbEL3453.EL3453.MDP5001_341_Input/MDP5001_341_Total_Basic_Calculated_Error_Current <-> Total Basic/Calculated Error Current
//     PlcTask Inputs/PRG_LVCP2_PowerMeasurement.fbEL3453.EL3453.MDP5001_341_Input/MDP5001_341_Total_Basic_Frequency <-> Total Basic/Frequency
//     PlcTask Inputs/PRG_LVCP2_PowerMeasurement.fbEL3453.EL3453.MDP5001_341_Input/MDP5001_341_Total_Basic_Neutral_Line_Current <-> Total Basic/Neutral Line Current
//     PlcTask Inputs/PRG_LVCP2_PowerMeasurement.fbEL3453.EL3453.MDP5001_341_Input/MDP5001_341_Total_Basic_Power_Factor <-> Total Basic/Power Factor
//     PlcTask Inputs/PRG_LVCP2_PowerMeasurement.fbEL3453.EL3453.MDP5001_341_Input/MDP5001_341_Total_Basic_ROCOF <-> Total Basic/ROCOF
//     PlcTask Inputs/PRG_LVCP2_PowerMeasurement.fbEL3453.EL3453.MDP5001_341_Input/MDP5001_341_Total_Status_Active_Power_Guard_Error <-> Total Status/Active Power Guard Error
//     PlcTask Inputs/PRG_LVCP2_PowerMeasurement.fbEL3453.EL3453.MDP5001_341_Input/MDP5001_341_Total_Status_Active_Power_Guard_Warning <-> Total Status/Active Power Guard Warning
//     PlcTask Inputs/PRG_LVCP2_PowerMeasurement.fbEL3453.EL3453.MDP5001_341_Input/MDP5001_341_Total_Status_Apparent_Power_Guard_Error <-> Total Status/Apparent Power Guard Error
//     PlcTask Inputs/PRG_LVCP2_PowerMeasurement.fbEL3453.EL3453.MDP5001_341_Input/MDP5001_341_Total_Status_Apparent_Power_Guard_Warning <-> Total Status/Apparent Power Guard Warning
//     PlcTask Inputs/PRG_LVCP2_PowerMeasurement.fbEL3453.EL3453.MDP5001_341_Input/MDP5001_341_Total_Status_Frequency_Guard_Error <-> Total Status/Frequency Guard Error
//     PlcTask Inputs/PRG_LVCP2_PowerMeasurement.fbEL3453.EL3453.MDP5001_341_Input/MDP5001_341_Total_Status_Frequency_Guard_Warning <-> Total Status/Frequency Guard Warning
//     PlcTask Inputs/PRG_LVCP2_PowerMeasurement.fbEL3453.EL3453.MDP5001_341_Input/MDP5001_341_Total_Status_Grid_Direction <-> Total Status/Grid Direction
//     PlcTask Inputs/PRG_LVCP2_PowerMeasurement.fbEL3453.EL3453.MDP5001_341_Input/MDP5001_341_Total_Status_Neutral_Current_Guard_Error <-> Total Status/Neutral Current Guard Error
//     PlcTask Inputs/PRG_LVCP2_PowerMeasurement.fbEL3453.EL3453.MDP5001_341_Input/MDP5001_341_Total_Status_Neutral_Current_Guard_Warning <-> Total Status/Neutral Current Guard Warning
//     PlcTask Inputs/PRG_LVCP2_PowerMeasurement.fbEL3453.EL3453.MDP5001_341_Input/MDP5001_341_Total_Status_Power_Quality_Factor <-> Total Status/Power Quality Factor
//     PlcTask Inputs/PRG_LVCP2_PowerMeasurement.fbEL3453.EL3453.MDP5001_341_Input/MDP5001_341_Total_Status_Power_Quality_Guard_Error <-> Total Status/Power Quality Guard Error
//     PlcTask Inputs/PRG_LVCP2_PowerMeasurement.fbEL3453.EL3453.MDP5001_341_Input/MDP5001_341_Total_Status_Power_Quality_Guard_Warning <-> Total Status/Power Quality Guard Warning
//     PlcTask Inputs/PRG_LVCP2_PowerMeasurement.fbEL3453.EL3453.MDP5001_341_Input/MDP5001_341_Total_Status_System_State <-> Total Status/System State
//     PlcTask Inputs/PRG_LVCP2_PowerMeasurement.fbEL3453.EL3453.MDP5001_341_Input/MDP5001_341_Total_Status_TxPDO_State <-> Total Status/TxPDO State
//     PlcTask Inputs/PRG_LVCP2_PowerMeasurement.fbEL3453.EL3453.MDP5001_341_Input/MDP5001_341_Total_Status_TxPDO_Toggle <-> Total Status/TxPDO Toggle
//     PlcTask Inputs/PRG_LVCP2_PowerMeasurement.fbEL3453.EL3453.MDP5001_341_Input/MDP5001_341_Total_Variant_Value_In_Index_1_REAL <-> Total Variant Value In/Index 1 REAL
//     PlcTask Inputs/PRG_LVCP2_PowerMeasurement.fbEL3453.EL3453.MDP5001_341_Input/MDP5001_341_Total_Variant_Value_In_Index_2_REAL <-> Total Variant Value In/Index 2 REAL
//     PlcTask Inputs/PRG_LVCP2_PowerMeasurement.fbEL3453.EL3453.MDP5001_341_Input/MDP5001_341_Total_Variant_Value_In_Index_3_REAL <-> Total Variant Value In/Index 3 REAL
//     PlcTask Inputs/PRG_LVCP2_PowerMeasurement.fbEL3453.EL3453.MDP5001_341_Input/MDP5001_341_Total_Variant_Value_In_Index_4_ULINT <-> Total Variant Value In/Index 4 ULINT
//     PlcTask Inputs/PRG_LVCP2_PowerMeasurement.fbEL3453.EL3453.MDP5001_341_Input/MDP5001_341_Total_Variant_Value_In_TxPDO_Toggle <-> Total Variant Value In/TxPDO Toggle
//     PlcTask Inputs/PRG_LVCP2_PowerMeasurement.fbEL3453.EL3453.MDP5001_341_Input/MDP5001_341_Total_Variant_Value_In_Value_1_REAL <-> Total Variant Value In/Value 1 REAL
//     PlcTask Inputs/PRG_LVCP2_PowerMeasurement.fbEL3453.EL3453.MDP5001_341_Input/MDP5001_341_Total_Variant_Value_In_Value_2_REAL <-> Total Variant Value In/Value 2 REAL
//     PlcTask Inputs/PRG_LVCP2_PowerMeasurement.fbEL3453.EL3453.MDP5001_341_Input/MDP5001_341_Total_Variant_Value_In_Value_3_REAL <-> Total Variant Value In/Value 3 REAL
//     PlcTask Inputs/PRG_LVCP2_PowerMeasurement.fbEL3453.EL3453.MDP5001_341_Input/MDP5001_341_Total_Variant_Value_In_Value_4_ULINT <-> Total Variant Value In/Value 4 ULINT
//     PlcTask Outputs/PRG_LVCP2_PowerMeasurement.fbEL3453.EL3453.MDP5001_341_Output/MDP5001_341_Total_Variant_Value_Out_Index_1_REAL <-> Total Variant Value Out/Index 1 REAL
//     PlcTask Outputs/PRG_LVCP2_PowerMeasurement.fbEL3453.EL3453.MDP5001_341_Output/MDP5001_341_Total_Variant_Value_Out_Index_2_REAL <-> Total Variant Value Out/Index 2 REAL
//     PlcTask Outputs/PRG_LVCP2_PowerMeasurement.fbEL3453.EL3453.MDP5001_341_Output/MDP5001_341_Total_Variant_Value_Out_Index_3_REAL <-> Total Variant Value Out/Index 3 REAL
//     PlcTask Outputs/PRG_LVCP2_PowerMeasurement.fbEL3453.EL3453.MDP5001_341_Output/MDP5001_341_Total_Variant_Value_Out_Index_4_ULINT <-> Total Variant Value Out/Index 4 ULINT
//   PLC/PLC Instance <-> Device 1 (EtherCAT)/+EP7-11CP1 (EK1100)/+EP7-11DI1 (EL1809)
//     PlcTask Inputs/GVL_Alarm.EP7_3X2_24VDC_OK <-> Channel 1/Input
//     PlcTask Inputs/GVL_Alarm.EP7_UPS_24VDC_OK <-> Channel 2/Input
//     PlcTask Inputs/PRG_LVCP2_Group{1..6}.stContactor_IO.bFeedback <-> Channel {6..16 step 2}/Input  (6 links)
//     PlcTask Inputs/PRG_LVCP2_Group{1..5}.stContactor_IO.bPLCControl <-> Channel {7..15 step 2}/Input  (5 links)
//     PlcTask Inputs/PRG_LVCP2_MainDisconnector.stDisconnectorIO.bLimitOff <-> Channel 4/Input
//     PlcTask Inputs/PRG_LVCP2_MainDisconnector.stDisconnectorIO.bLimitOn <-> Channel 3/Input
//     PlcTask Inputs/PRG_LVCP2_MainDisconnector.stDisconnectorIO.bPLCControl <-> Channel 5/Input
//   PLC/PLC Instance <-> Device 1 (EtherCAT)/+EP7-11CP1 (EK1100)/+EP7-11DI2 (EL1809)
//     PlcTask Inputs/PRG_LVCP2_Group{7..10}.stContactor_IO.bFeedback <-> Channel {2..8 step 2}/Input  (4 links)
//     PlcTask Inputs/PRG_LVCP2_Group{6..10}.stContactor_IO.bPLCControl <-> Channel {1..9 step 2}/Input  (5 links)
//   PLC/PLC Instance <-> Device 1 (EtherCAT)/+EP7-11CP1 (EK1100)/+EP7-11DQ1 (EL2809-0015)
//     PlcTask Outputs/PRG_LVCP2_Group{1..10}.stContactor_IO.bOutput <-> Channel {3..12}/Output  (10 links)
//     PlcTask Outputs/PRG_LVCP2_MainDisconnector.stDisconnectorIO.bContactorOff_Out <-> Channel 2/Output
//     PlcTask Outputs/PRG_LVCP2_MainDisconnector.stDisconnectorIO.bContactorOn_Out <-> Channel 1/Output
//   PLC/PLC Instance <-> Device 1 (EtherCAT)/+EP8-11CP1 (EK1100)/+EP8-11DI1 (EL1809)
//     PlcTask Inputs/GVL_Alarm.EP8_3X2_24VDC_OK <-> Channel 1/Input
//     PlcTask Inputs/GVL_Alarm.EP8_UPS_24VDC_OK <-> Channel 2/Input
//   PLC/PLC Instance <-> Device 1 (EtherCAT)/+EP9-5CP5 (EK1100)/+EP9-5DI1 (EL1809)
//     PlcTask Inputs/GVL_Alarm.EP9_3X2_24VDC_OK <-> Channel 1/Input
//     PlcTask Inputs/GVL_Alarm.EP9_UPS_24VDC_OK <-> Channel 2/Input
//     PlcTask Inputs/PRG_HVCP3_10CB1.stDisconnectorIO.bEarthSwitchOff <-> Channel 7/Input
//     PlcTask Inputs/PRG_HVCP3_10CB1.stDisconnectorIO.bEarthSwitchOn <-> Channel 6/Input
//     PlcTask Inputs/PRG_HVCP3_10CB1.stDisconnectorIO.bLimitOff <-> Channel 4/Input
//     PlcTask Inputs/PRG_HVCP3_12CB1.stDisconnectorIO.bLimitOff <-> Channel 9/Input
//     PlcTask Inputs/PRG_HVCP3_14CB1.stDisconnectorIO.bLimitOff <-> Channel 12/Input
//     PlcTask Inputs/PRG_HVCP3_16CB1.stDisconnectorIO.bLimitOff <-> Channel 15/Input
//     PlcTask Inputs/PRG_HVCP3_10CB1.stDisconnectorIO.bLimitOn <-> Channel 3/Input
//     PlcTask Inputs/PRG_HVCP3_12CB1.stDisconnectorIO.bLimitOn <-> Channel 8/Input
//     PlcTask Inputs/PRG_HVCP3_14CB1.stDisconnectorIO.bLimitOn <-> Channel 11/Input
//     PlcTask Inputs/PRG_HVCP3_16CB1.stDisconnectorIO.bLimitOn <-> Channel 14/Input
//     PlcTask Inputs/PRG_HVCP3_10CB1.stDisconnectorIO.bPLCControl <-> Channel 5/Input
//     PlcTask Inputs/PRG_HVCP3_12CB1.stDisconnectorIO.bPLCControl <-> Channel 10/Input
//     PlcTask Inputs/PRG_HVCP3_14CB1.stDisconnectorIO.bPLCControl <-> Channel 13/Input
//     PlcTask Inputs/PRG_HVCP3_16CB1.stDisconnectorIO.bPLCControl <-> Channel 16/Input
//   PLC/PLC Instance <-> Device 1 (EtherCAT)/+EP9-5CP5 (EK1100)/+EP9-5DI2 (EL1809)
//     PlcTask Inputs/PRG_HVCP3_{18..26 step 2}CB1.stDisconnectorIO.bLimitOff <-> Channel {2..14 step 3}/Input  (5 links)
//     PlcTask Inputs/PRG_HVCP3_{18..28 step 2}CB1.stDisconnectorIO.bLimitOn <-> Channel {1..16 step 3}/Input  (6 links)
//     PlcTask Inputs/PRG_HVCP3_{18..26 step 2}CB1.stDisconnectorIO.bPLCControl <-> Channel {3..15 step 3}/Input  (5 links)
//   PLC/PLC Instance <-> Device 1 (EtherCAT)/+EP9-5CP5 (EK1100)/+EP9-5DI3 (EL1809)
//     PlcTask Inputs/PRG_HVCP3_{28..38 step 2}CB1.stDisconnectorIO.bLimitOff <-> Channel {1..16 step 3}/Input  (6 links)
//     PlcTask Inputs/PRG_HVCP3_{28..36 step 2}CB1.stDisconnectorIO.bPLCControl <-> Channel {2..14 step 3}/Input  (5 links)
//     PlcTask Inputs/PRG_HVCP3_{30..38 step 2}CB1.stDisconnectorIO.bLimitOn <-> Channel {3..15 step 3}/Input  (5 links)
//   PLC/PLC Instance <-> Device 1 (EtherCAT)/+EP9-5CP5 (EK1100)/+EP9-5DI4 (EL1809)
//     PlcTask Inputs/PRG_HVCP3_{38..48 step 2}CB1.stDisconnectorIO.bPLCControl <-> Channel {1..16 step 3}/Input  (6 links)
//     PlcTask Inputs/PRG_HVCP3_{40..48 step 2}CB1.stDisconnectorIO.bLimitOff <-> Channel {3..15 step 3}/Input  (5 links)
//     PlcTask Inputs/PRG_HVCP3_{40..48 step 2}CB1.stDisconnectorIO.bLimitOn <-> Channel {2..14 step 3}/Input  (5 links)
//   PLC/PLC Instance <-> Device 1 (EtherCAT)/+EP9-5CP5 (EK1100)/+EP9-5DI5 (EL1809)
//     PlcTask Inputs/PRG_HVCP3_{50..56 step 2}CB1.stDisconnectorIO.bLimitOff <-> Channel {2..11 step 3}/Input  (4 links)
//     PlcTask Inputs/PRG_HVCP3_{50..56 step 2}CB1.stDisconnectorIO.bLimitOn <-> Channel {1..10 step 3}/Input  (4 links)
//     PlcTask Inputs/PRG_HVCP3_{50..56 step 2}CB1.stDisconnectorIO.bPLCControl <-> Channel {3..12 step 3}/Input  (4 links)
//   PLC/PLC Instance <-> Device 1 (EtherCAT)/+EP9-5CP5 (EK1100)/+EP9-5DQ1 (EL2809)
//     PlcTask Outputs/PRG_HVCP3_{10..24 step 2}CB1.stDisconnectorIO.bContactorOff_Out <-> Channel {2..16 step 2}/Output  (8 links)
//     PlcTask Outputs/PRG_HVCP3_{10..24 step 2}CB1.stDisconnectorIO.bContactorOn_Out <-> Channel {1..15 step 2}/Output  (8 links)
//   PLC/PLC Instance <-> Device 1 (EtherCAT)/+EP9-5CP5 (EK1100)/+EP9-5DQ2 (EL2809)
//     PlcTask Outputs/PRG_HVCP3_{26..40 step 2}CB1.stDisconnectorIO.bContactorOff_Out <-> Channel {2..16 step 2}/Output  (8 links)
//     PlcTask Outputs/PRG_HVCP3_{26..40 step 2}CB1.stDisconnectorIO.bContactorOn_Out <-> Channel {1..15 step 2}/Output  (8 links)
//   PLC/PLC Instance <-> Device 1 (EtherCAT)/+EP9-5CP5 (EK1100)/+EP9-5DQ3 (EL2809)
//     PlcTask Outputs/PRG_HVCP3_{42..56 step 2}CB1.stDisconnectorIO.bContactorOff_Out <-> Channel {2..16 step 2}/Output  (8 links)
//     PlcTask Outputs/PRG_HVCP3_{42..56 step 2}CB1.stDisconnectorIO.bContactorOn_Out <-> Channel {1..15 step 2}/Output  (8 links)

CONFIGURATION PLC
    RESOURCE PLC ON TwinCAT3
        TASK PlcTask(INTERVAL := T#10ms, PRIORITY := 20);
        PROGRAM MAIN WITH PlcTask : MAIN;
    END_RESOURCE
END_CONFIGURATION

// ---- POUs/EL3453/stEL3453.TcDUT
TYPE stEL3453 :
STRUCT
	Lx 			: ARRAY[1..3] OF stEL3453_ch;
	Total 		: stEL3453_tot;
END_STRUCT
END_TYPE

// ---- POUs/EL3453/stEL3453_ch.TcDUT
TYPE stEL3453_ch :
STRUCT
	fULrms		: REAL;  //[V]
	fUL_peak 	: REAL;  //[V]
	ulUL_ZC		: ULINT;  //[ns]
	fULrms_min	: REAL; //[V]
	fULrms_max	: REAL; //[V]
	fUL_THD		: REAL; //[% of fundamental rms]
	fULrms_fund	: REAL; //[V]
	fUL_harm	: ARRAY [0..63] OF REAL; //[% of fundamental rms]
	fUL_harmrf	: REAL;  //[Hz]
	
	fIrms 		: REAL; //[A]
	fI_peak		: REAL; //[A]
	ulI_ZC		: ULINT; //[ns]
	fIrms_min	: REAL;  //[A]
	fIrms_max	: REAL;  //[A]
	fI_THD		: REAL;  //[% of fundamental rms]
	fI_TDD		: REAL;  //[% of max rms]
	fIrms_fund	: REAL;  //[A]
	fIL_harm	: ARRAY [0..63] OF REAL;  //[% of fundamental rms]
	fIL_harmrf	: REAL;  //[Hz]
	
	fFreq		: REAL; //[Hz]
	fPhi		: REAL; //[°]
	fCosPhi		: REAL; //[ ]
	fPF			: REAL; //[ ]
	
	fP			: REAL; //[W]
	fP_avg		: REAL; //[W]
	fP_min		: REAL; //[W]
	fP_max		: REAL; //[W]
	fP_fund		: REAL; //[W]
	
	fS			: REAL; //[VA]
	fS_avg		: REAL; //[VA]
	fS_min		: REAL; //[VA]
	fS_max		: REAL; //[VA]
	fS_fund		: REAL; //[VA]
	
	fQ			: REAL; //[VAR]
	fQ_avg		: REAL; //[VAR]
	fQ_min		: REAL; //[VAR]
	fQ_max		: REAL; //[VAR]
	fQ_fund		: REAL; //[VAR]
	
	lEP 		: LINT;  //[mWh]
	ulEP_pos	: ULINT; //[mWh]
	ulEP_neg	: ULINT; //[mWh]
	
	lES 		: LINT; //[mVAh]
	ulES_pos	: ULINT; //[mVAh]
	ulES_neg	: ULINT; //[mVAh]
	
	lEQ			: LINT; //[mVArh]
	ulEQ_pos	: ULINT; //[mVArh]
	ulEQ_neg	: ULINT; //[mVArh]
	
	lEP_fund		: LINT; //[mWh]
	ulEP_fund_pos	: ULINT; //[mWh]
	ulEP_fund_neg	: ULINT; //[mWh]
	
	lES_fund 		: LINT; //[mVAh]
	ulES_fund_pos	: ULINT; //[mVAh]
	ulES_fund_neg	: ULINT; //[mVAh]
	
	lEQ_fund		: LINT; //[mVArh]
	ulEQ_fund_pos	: ULINT; //[mVArh]
	ulEQ_fund_neg	: ULINT; //[mVArh]
	
	
END_STRUCT
END_TYPE

// ---- POUs/EL3453/stEL3453_tot.TcDUT
TYPE stEL3453_tot :
STRUCT
	
	fInrms				: REAL;	//[A]
	fIerrrmsCalc		: REAL; //[A]
	fPF					: REAL; //[ ]
	fFreq				: REAL; //[Hz]
	
	fUL12				: REAL; //[V]
	fUL23				: REAL; //[V]
	fUL31				: REAL; //[V]
	
	fP					: REAL; //[W]
	fP_avg				: REAL; //[W]
	fP_min 				: REAL; //[W]
	fP_max				: REAL; //[W]
	
	fS					: REAL; //[VA]
	fS_avg				: REAL; //[VA]
	fS_min	 			: REAL; //[VA]
	fS_max				: REAL; //[VA]
	
	fQtot				: REAL; //[VAR]
	fQtot_avg			: REAL; //[VAR]
	fQtot_min 			: REAL; //[VAR]
	fQtot_max			: REAL; //[VAR]
	
	lEP 				: LINT; //[mWh]
	ulEP_pos			: ULINT; //[mWh]
	ulEP_neg			: ULINT; //[mWh]
	 lEP_int			: LINT; //[mWh]
	ulEP_int_pos		: ULINT; //[mWh]
	ulEP_int_neg		: ULINT; //[mWh]
	
	 lEP_fund 			: LINT; //[mWh]
	ulEP_fund_pos		: ULINT; //[mWh]
	ulEP_fund_neg		: ULINT; //[mWh]
	 lEP_fund_int		: LINT; //[mWh]
	ulEP_fund_int_pos	: ULINT; //[mWh]
	ulEP_fund_int_neg	: ULINT; //[mWh]
	
	 lES 				: LINT; //[mVAh]
	ulES_pos			: ULINT; //[mVAh]
	ulES_neg			: ULINT; //[mVAh]
	 lES_int			: LINT; //[mVAh]
	ulES_int_pos		: ULINT; //[mVAh]
	ulES_int_neg		: ULINT; //[mVAh]
	
	 lES_fund 			: LINT; //[mVAh]
	ulES_fund_pos		: ULINT; //[mVAh]
	ulES_fund_neg		: ULINT; //[mVAh]
	 lES_fund_int		: LINT; //[mVAh]
	ulES_fund_int_pos	: ULINT; //[mVAh]
	ulES_fund_int_neg	: ULINT; //[mVAh]
	
	 lEQ				: LINT; //[mVARh]
	ulEQ_pos			: ULINT; //[mVARh]
	ulEQ_neg			: ULINT; //[mVARh]
	 lEQ_int			: LINT; //[mVARh]
	ulEQ_int_pos		: ULINT; //[mVARh]
	ulEQ_int_neg		: ULINT; //[mVARh]
			
	 lEQ_fund 			: LINT; //[mVARh]
	ulEQ_fund_pos		: ULINT; //[mVARh]
	ulEQ_fund_neg		: ULINT; //[mVARh]
	 lEQ_fund_int		: LINT; //[mVARh]
	ulEQ_fund_int_pos	: ULINT; //[mVARh]
	ulEQ_fund_int_neg	: ULINT; //[mVARh]
	
	fPhiL1L2			: REAL; //[°]
	fPhiL1L3			: REAL; //[°]
	fUnbalance			: REAL; //[%]
	
	fPQF				: REAL; //[%]
	fPQF_avg			: REAL; //[%]
	fPQF_min			: REAL; //[%]
	fPQF_max			: REAL; //[%]
	
	fP_fund				: REAL; //[W]
	fP_fund_avg			: REAL; //[W] 
	fP_fund_min			: REAL; //[W]
	fP_fund_max			: REAL; //[W]
	
	fS_fund				: REAL; //[VA]
	fS_fund_avg			: REAL; //[VA]
	fS_fund_min			: REAL; //[VA]
	fS_fund_max			: REAL; //[VA]
	
	fQ_fund				: REAL;	//[VAR]
	fQ_fund_avg			: REAL; //[VAR]
	fQ_fund_min			: REAL; //[VAR]
	fQ_fund_max			: REAL; //[VAR]
	
END_STRUCT
END_TYPE

// ---- _ES/11_Disconnector/Enum/E_DisconnectorControlMode.TcTLEO
TYPE E_DisconnectorControlMode :
(
    MANUAL := 0,     // Manuel kontrol - Lokal butonlar
    AUTO := 1,       // Otomatik kontrol - PLC lojiği
    REMOTE := 2      // Uzaktan kontrol - SCADA/HMI
);
END_TYPE

// ---- _ES/11_Disconnector/Enum/E_DisconnectorFault.TcTLEO
TYPE E_DisconnectorFault :
(
    NONE := 0,                  // Arıza yok
    THERMAL := 1,               // Termik arıza
    CONTACTOR_ON := 2,          // ON kontaktör geri bildirim hatası
    CONTACTOR_OFF := 3,         // OFF kontaktör geri bildirim hatası
    MOTION_TIMEOUT := 4,        // Hareket zaman aşımı
    BOTH_LIMITS := 5,           // Her iki limit aktif
    INTERLOCK := 6,             // Toprak bıçağı interlock hatası
    EARTH_SWITCH := 7           // Toprak bıçağı senkronizasyon hatası
);
END_TYPE

// ---- _ES/11_Disconnector/Enum/E_DisconnectorPosition.TcTLEO
TYPE E_DisconnectorPosition : 
(
    UNDEFINED := 0,
    OFF := 1,
    TURNING_ON := 2,
    ON := 3,
    TURNING_OFF := 4,
    FAULT := 5
);
END_TYPE

// ---- _ES/11_Disconnector/Enum/E_DisconnectorStatus.TcTLEO
TYPE E_DisconnectorStatus :
(
    READY := 0,          // Hazır
    OPERATING := 1,      // Hareket halinde
    INTERLOCKED := 2,    // Interlock aktif
    FAULTED := 3,        // Arızalı
    NO_CONTROL := 4,     // PLC kontrol yok
    MAINTENANCE := 5     // Bakım gerekli
);
END_TYPE

// ---- _ES/11_Disconnector/Structure/ST_DisconnectorCommand.TcDUT
TYPE ST_DisconnectorCommand :
STRUCT
    eControlMode: E_DisconnectorControlMode;    // Kontrol modu seçimi
    bAutoOnCmd: BOOL;                           // Otomatik ON komutu
    bAutoOffCmd: BOOL;                          // Otomatik OFF komutu
    bResetFault: BOOL;                          // Hata reset sinyali
    bResetStatistics: BOOL;                     // İstatistik reset sinyali
    bManualOnCmd: BOOL;                         // Manuel ON komutu
    bManualOffCmd: BOOL;                        // Manuel OFF komutu
    bStop: BOOL;                                // Hareketi durdur komutu
END_STRUCT
END_TYPE

// ---- _ES/11_Disconnector/Structure/ST_DisconnectorConfig.TcDUT
TYPE ST_DisconnectorConfig :
STRUCT
    // Kimlik Bilgileri
    sProjectCode: STRING[20] := '';             // Proje kodu (örn: +EP1-23D1)
    sProductCode: STRING[50] := '';             // Ürün kodu/modeli
    
    // Elektriksel Özellikler
    rRatedCurrent: REAL := 0.0;                 // Nominal akım (A)
    rRatedVoltage: REAL := 0.0;                 // Nominal gerilim (kV)
    nPhaseCount: INT := 3;                      // Faz sayısı (1 veya 3)
    bGrounded: BOOL := FALSE;                   // Topraklı tip mi?
    
    // Operasyonel Parametreler
    tMotionTimeout: TIME := T#30S;              // Hareket zaman aşımı
    tContactorDelay: TIME := T#500MS;           // Kontaktör geri bildirim gecikmesi
    bContactorFeedbackRequired: BOOL := FALSE;   // Kontaktör geri bildirimi gerekli mi?
    bEarthSwitchExists: BOOL;                   // Toprak bıçağı mevcut mu?
    bInterlockEnable: BOOL;                     // Interlock kontrolü aktif mi?
    dwOperationLimit: DWORD := 10000;           // Bakım operasyon limiti
END_STRUCT
END_TYPE

// ---- _ES/11_Disconnector/Structure/ST_DisconnectorHMI.TcDUT
TYPE ST_DisconnectorHMI :
STRUCT
    stCommand: ST_DisconnectorCommand;          // Komutlar
    stStatus: ST_DisconnectorStatus;            // Durum bilgileri
    stConfig: ST_DisconnectorConfig;            // Konfigürasyon
    stStatistics: ST_DisconnectorStatistics;    // İstatistik verileri
END_STRUCT
END_TYPE

// ---- _ES/11_Disconnector/Structure/ST_DisconnectorIO.TcDUT
TYPE ST_DisconnectorIO :
STRUCT
    // Giriş Sinyalleri
    bContactorOn_FB AT %I*: BOOL;      // ON kontaktörü geri bildirimi
    bContactorOff_FB AT %I*: BOOL;     // OFF kontaktörü geri bildirimi
    bLimitOn AT %I*: BOOL;             // ON pozisyon limit switch
    bLimitOff AT %I*: BOOL;            // OFF pozisyon limit switch
    bThermalFault AT %I*: BOOL;        // Motor termik koruma arızası
    bEarthSwitchOn AT %I*: BOOL;       // Toprak bıçağı ON pozisyonu
    bEarthSwitchOff AT %I*: BOOL;      // Toprak bıçağı OFF pozisyonu
    bPLCControl AT %I*: BOOL;          // PLC kontrol seçici
    
    // Çıkış Sinyalleri
    bContactorOn_Out AT %Q*: BOOL;     // ON kontaktörü sürme
    bContactorOff_Out AT %Q*: BOOL;    // OFF kontaktörü sürme
END_STRUCT
END_TYPE

// ---- _ES/11_Disconnector/Structure/ST_DisconnectorOperationRecord.TcDUT
TYPE ST_DisconnectorOperationRecord :
STRUCT
    dtTimestamp: DATE_AND_TIME;                 // İşlem zamanı
    eOperation: E_DisconnectorPosition;            // İşlem tipi (ON/OFF/FAULT)
    eControlMode: E_DisconnectorControlMode;    // Kontrol modu
    tTransitionTime: TIME;                      // Geçiş süresi
    eFaultCode: E_DisconnectorFault;            // Arıza kodu (varsa)
    nDisconnectorID: INT;                       // Ayırıcı ID
END_STRUCT
END_TYPE

// ---- _ES/11_Disconnector/Structure/ST_DisconnectorStatistics.TcDUT
TYPE ST_DisconnectorStatistics :
STRUCT
    // Çalışma Sayaçları
    dwOnCount: DWORD;                           // Toplam ON sayısı
    dwOffCount: DWORD;                          // Toplam OFF sayısı
    dwOperationCount: DWORD;                    // Toplam operasyon sayısı
    
    // Son İşlem Bilgisi (SQL buffer)
    stLastOperation: ST_DisconnectorOperationRecord;  // SQL'e yazılacak son işlem
    bNewOperationFlag: BOOL;                    // Yeni işlem var, SQL'e yaz
    
    // Arıza İstatistikleri
    dwTotalFaultCount: DWORD;                   // Toplam arıza sayısı
    dwThermalFaultCount: DWORD;                 // Termik arıza sayısı
    dwMotionTimeoutCount: DWORD;                // Hareket zaman aşımı sayısı
    dwContactorFaultCount: DWORD;               // Kontaktör arıza sayısı
    dwInterlockFaultCount: DWORD;               // Interlock arıza sayısı
    
    // Performans Verileri
    tLastOnTransitionTime: TIME;                // Son ON geçiş süresi
    tLastOffTransitionTime: TIME;               // Son OFF geçiş süresi
    tMaxOnTransitionTime: TIME;                 // Maksimum ON geçiş süresi
    tMaxOffTransitionTime: TIME;                // Maksimum OFF geçiş süresi
    
    // Bakım Bilgileri
    bMaintenanceRequired: BOOL;                 // Bakım gerekli
    dwRemainingOperations: DWORD;               // Kalan operasyon sayısı
END_STRUCT
END_TYPE

// ---- _ES/11_Disconnector/Structure/ST_DisconnectorStatus.TcDUT
TYPE ST_DisconnectorStatus :
STRUCT
    ePosition: E_DisconnectorPosition;          // Ayırıcı fiziksel pozisyonu
    eEarthSwitchPosition: E_DisconnectorPosition; // Toprak bıçağı pozisyonu
    eStatus: E_DisconnectorStatus;              // Operasyonel durum
    eActiveMode: E_DisconnectorControlMode;     // Aktif kontrol modu
    bTurningOn: BOOL;                           // ON'a geçiyor durumu
    bTurningOff: BOOL;                          // OFF'a geçiyor durumu
    bFaultActive: BOOL;                         // Arıza durumu
    eFaultCode: E_DisconnectorFault;            // Arıza kodu
    bPLCControlActive: BOOL;                    // PLC kontrol durumu
    bContactorOn_Out: BOOL;                     // ON kontaktörü sürme
    bContactorOff_Out: BOOL;                    // OFF kontaktörü sürme
    wsStatusText: WSTRING(100);                 // Durum açıklama metni
END_STRUCT
END_TYPE

// ---- _ES/12_Contactor/Enum/E_ContactorControlMode.TcTLEO
TYPE E_ContactorControlMode :
(
    MANUAL := 0,        // Manuel kontrol - Lokal butonlar
    AUTO := 1,          // Otomatik kontrol - PLC lojiği
    REMOTE := 2         // Uzaktan kontrol - SCADA/HMI
);
END_TYPE

// ---- _ES/12_Contactor/Enum/E_ContactorFault.TcTLEO
TYPE E_ContactorFault :
(
    NONE := 0,          // Arıza yok
    FEEDBACK := 1,      // Geri besleme hatası
    WELDED := 2,        // Kontak yapışması
    COIL := 3           // Bobin arızası
);
END_TYPE

// ---- _ES/12_Contactor/Enum/E_ContactorPosition.TcTLEO
TYPE E_ContactorPosition :
(
    UNDEFINED := 0,     // Belirsiz durum (ilk çalıştırma)
    OFF := 1,           // Kontaktör kapalı
    ON := 2             // Kontaktör açık
);
END_TYPE

// ---- _ES/12_Contactor/Enum/E_ContactorStatus.TcTLEO
TYPE E_ContactorStatus :
(
    READY := 0,         // Hazır
    OPERATING := 1,     // Çalışıyor
    INTERLOCKED := 2,   // Interlock aktif
    FAULTED := 3,       // Arızalı
    NO_CONTROL := 4,    // PLC kontrol yok
    MAINTENANCE := 5    // Bakım gerekli
);
END_TYPE

// ---- _ES/12_Contactor/Structure/ST_ContactorCommand.TcDUT
TYPE ST_ContactorCommand :
STRUCT
    eControlMode: E_ContactorControlMode;       // Kontrol modu seçimi
    bAutoOnCmd: BOOL;                          // Otomatik ON komutu
    bAutoOffCmd: BOOL;                         // Otomatik OFF komutu
    bManualOnCmd: BOOL;                        // Manuel ON komutu
    bManualOffCmd: BOOL;                       // Manuel OFF komutu
    bResetFault: BOOL;                         // Hata reset sinyali
    bResetStatistics: BOOL;                    // İstatistik reset sinyali
END_STRUCT
END_TYPE

// ---- _ES/12_Contactor/Structure/ST_ContactorConfig.TcDUT
TYPE ST_ContactorConfig :
STRUCT
    // Kimlik Bilgileri
    sProjectCode: STRING[20] := '';             // Proje kodu (örn: +EP1-K1)
    sProductCode: STRING[50] := '';             // Ürün kodu/modeli
    
    // Elektriksel Özellikler
    rRatedCurrent: REAL := 0.0;                 // Nominal akım (A)
    rRatedVoltage: REAL := 0.0;                 // Nominal gerilim (V)
    nPhaseCount: INT := 3;                      // Faz sayısı (1 veya 3)
    
    // Operasyonel Parametreler
    tFeedbackDelay: TIME := T#500MS;            // Geri bildirim gecikmesi
    tWeldedDelay: TIME := T#2S;                 // Yapışma kontrolü gecikmesi
    bFeedbackRequired: BOOL := FALSE;            // Geri bildirim gerekli mi?
    dwOperationLimit: DWORD := 100000;          // Bakım operasyon limiti
END_STRUCT
END_TYPE

// ---- _ES/12_Contactor/Structure/ST_ContactorHMI.TcDUT
TYPE ST_ContactorHMI :
STRUCT
    stCommand: ST_ContactorCommand;             // Komutlar
    stStatus: ST_ContactorStatus;               // Durum bilgileri
    stConfig: ST_ContactorConfig;               // Konfigürasyon
    stStatistics: ST_ContactorStatistics;       // İstatistik verileri
END_STRUCT
END_TYPE

// ---- _ES/12_Contactor/Structure/ST_ContactorIO.TcDUT
TYPE ST_ContactorIO :
STRUCT
    // Giriş Sinyalleri
    bFeedback AT %I*: BOOL;         // Kontaktör yardımcı kontak geri bildirimi
    bPLCControl AT %I*: BOOL;       // PLC kontrol seçici
    
    // Çıkış Sinyalleri
    bOutput AT %Q*: BOOL;           // Kontaktör bobini
END_STRUCT
END_TYPE

// ---- _ES/12_Contactor/Structure/ST_ContactorOperationRecord.TcDUT
TYPE ST_ContactorOperationRecord :
STRUCT
    dtTimestamp: DATE_AND_TIME;                 // İşlem zamanı
    eOperation: E_ContactorPosition;            // İşlem tipi (ON/OFF)
    eControlMode: E_ContactorControlMode;        // Kontrol modu
    eFaultCode: E_ContactorFault;               // Arıza kodu (varsa)
    nContactorID: INT;                          // Kontaktör ID
END_STRUCT
END_TYPE

// ---- _ES/12_Contactor/Structure/ST_ContactorStatistics.TcDUT
TYPE ST_ContactorStatistics :
STRUCT
    // Çalışma Sayaçları
    dwOnCount: DWORD;                           // Toplam ON sayısı
    dwOffCount: DWORD;                          // Toplam OFF sayısı
    dwOperationCount: DWORD;                    // Toplam operasyon sayısı
    
    // Son İşlem Bilgisi (SQL buffer)
    stLastOperation: ST_ContactorOperationRecord; // SQL'e yazılacak son işlem
    bNewOperationFlag: BOOL;                    // Yeni işlem var, SQL'e yaz
    
    // Arıza İstatistikleri
    dwTotalFaultCount: DWORD;                   // Toplam arıza sayısı
    dwFeedbackFaultCount: DWORD;                // Geri besleme arıza sayısı
    dwWeldedFaultCount: DWORD;                  // Yapışma arıza sayısı
    
    // Bakım Bilgileri
    bMaintenanceRequired: BOOL;                 // Bakım gerekli
    dwRemainingOperations: DWORD;               // Kalan operasyon sayısı
END_STRUCT
END_TYPE

// ---- _ES/12_Contactor/Structure/ST_ContactorStatus.TcDUT
TYPE ST_ContactorStatus :
STRUCT
    ePosition: E_ContactorPosition;             // Kontaktör pozisyonu
    eStatus: E_ContactorStatus;                 // Operasyonel durum
    eActiveMode: E_ContactorControlMode;        // Aktif kontrol modu
    bFaultActive: BOOL;                         // Arıza durumu
    eFaultCode: E_ContactorFault;                // Arıza kodu
    bPLCControlActive: BOOL;                    // PLC kontrol durumu
    bOutput: BOOL;                              // Kontaktör çıkışı
    wsStatusText: WSTRING(100);                 // Durum açıklama metni
END_STRUCT
END_TYPE

// ---- _ES/13_CircuitBreaker/Enum/E_CircuitBreakerControlMode.TcTLEO
TYPE E_CircuitBreakerControlMode :
(
    MANUAL := 0,        // Manuel kontrol
    AUTO := 1,          // Otomatik kontrol
    REMOTE := 2         // Uzaktan kontrol
);
END_TYPE

// ---- _ES/13_CircuitBreaker/Enum/E_CircuitBreakerFault.TcTLEO
TYPE E_CircuitBreakerFault :
(
    NONE := 0,              // Arıza yok
    SPRING_CHARGE := 1,     // Yay kurma arızası
    FEEDBACK := 2,          // Geri besleme hatası
    MOTION_TIMEOUT := 3,    // Hareket zaman aşımı
    TRIP_COIL := 4,         // Trip bobini arızası
    CONTROL_VOLTAGE := 5    // Kontrol gerilimi arızası
);
END_TYPE

// ---- _ES/13_CircuitBreaker/Enum/E_CircuitBreakerPosition.TcTLEO
TYPE E_CircuitBreakerPosition :
(
    UNDEFINED := 0,     // Belirsiz durum
    OFF := 1,           // OFF pozisyonu
    ON := 2,            // ON pozisyonu
    TRIPPED := 3        // TRIP pozisyonu
);
END_TYPE

// ---- _ES/13_CircuitBreaker/Enum/E_CircuitBreakerStatus.TcTLEO
TYPE E_CircuitBreakerStatus :
(
    READY := 0,         // Hazır
    OPERATING := 1,     // Hareket halinde
    INTERLOCKED := 2,   // Interlock aktif
    FAULTED := 3,       // Arızalı
    TRIPPED := 4,       // Trip durumunda
    NO_CONTROL := 5,    // PLC kontrol yok
    MAINTENANCE := 6    // Bakım gerekli
);
END_TYPE

// ---- _ES/13_CircuitBreaker/Structure/ST_CircuitBreakerCommand.TcDUT
TYPE ST_CircuitBreakerCommand :
STRUCT
    eControlMode: E_CircuitBreakerControlMode;  // Kontrol modu seçimi
    bAutoOnCmd: BOOL;                           // Otomatik ON komutu
    bAutoOffCmd: BOOL;                          // Otomatik OFF komutu
    bManualOnCmd: BOOL;                         // Manuel ON komutu
    bManualOffCmd: BOOL;                        // Manuel OFF komutu
    bResetTrip: BOOL;                           // Trip reset komutu
    bResetFault: BOOL;                          // Hata reset sinyali
    bResetStatistics: BOOL;                     // İstatistik reset sinyali
END_STRUCT
END_TYPE

// ---- _ES/13_CircuitBreaker/Structure/ST_CircuitBreakerConfig.TcDUT
TYPE ST_CircuitBreakerConfig :
STRUCT
    // Kimlik Bilgileri
    sProjectCode: STRING[20] := '';             // Proje kodu (örn: +EP1-Q1)
    sProductCode: STRING[50] := '';             // Ürün kodu/modeli
    
    // Elektriksel Özellikler
    rRatedCurrent: REAL := 0.0;                 // Nominal akım (A)
    rRatedVoltage: REAL := 0.0;                 // Nominal gerilim (kV)
    nPhaseCount: INT := 3;                      // Faz sayısı (1 veya 3)
    
    // Operasyonel Parametreler
    tMotionTimeout: TIME := T#5S;               // Hareket zaman aşımı
    tSpringChargeTimeout: TIME := T#30S;        // Yay kurma zaman aşımı
    bSpringChargeRequired: BOOL := TRUE;        // Yay kurma gerekli mi?
    dwOperationLimit: DWORD := 10000;           // Bakım operasyon limiti
END_STRUCT
END_TYPE

// ---- _ES/13_CircuitBreaker/Structure/ST_CircuitBreakerHMI.TcDUT
TYPE ST_CircuitBreakerHMI :
STRUCT
    stCommand: ST_CircuitBreakerCommand;        // Komutlar
    stStatus: ST_CircuitBreakerStatus;          // Durum bilgileri
    stConfig: ST_CircuitBreakerConfig;          // Konfigürasyon
    stStatistics: ST_CircuitBreakerStatistics;  // İstatistik verileri
END_STRUCT
END_TYPE

// ---- _ES/13_CircuitBreaker/Structure/ST_CircuitBreakerIO.TcDUT
TYPE ST_CircuitBreakerIO :
STRUCT
    // Giriş Sinyalleri
    bPositionOn AT %I*: BOOL;           // ON pozisyon geri bildirimi
    bPositionOff AT %I*: BOOL;          // OFF pozisyon geri bildirimi
    bPositionTripped AT %I*: BOOL;      // TRIP pozisyon geri bildirimi
    bSpringCharged AT %I*: BOOL;        // Yay kurulu bilgisi
    bPLCControl AT %I*: BOOL;           // PLC kontrol seçici
    
    // Çıkış Sinyalleri
    bOnCommand AT %Q*: BOOL;            // ON komutu
    bOffCommand AT %Q*: BOOL;           // OFF komutu
END_STRUCT
END_TYPE

// ---- _ES/13_CircuitBreaker/Structure/ST_CircuitBreakerOperationRecord.TcDUT
TYPE ST_CircuitBreakerOperationRecord :
STRUCT
    dtTimestamp: DATE_AND_TIME;                 // İşlem zamanı
    eOperation: E_CircuitBreakerPosition;       // İşlem tipi (ON/OFF/TRIPPED)
    eControlMode: E_CircuitBreakerControlMode;  // Kontrol modu
    eFaultCode: E_CircuitBreakerFault;          // Arıza kodu (varsa)
    nBreakerID: INT;                            // Kesici ID
END_STRUCT
END_TYPE

// ---- _ES/13_CircuitBreaker/Structure/ST_CircuitBreakerStatistics.TcDUT
TYPE ST_CircuitBreakerStatistics :
STRUCT
    // Çalışma Sayaçları
    dwOnCount: DWORD;                           // Toplam ON sayısı
    dwOffCount: DWORD;                          // Toplam OFF sayısı
    dwTripCount: DWORD;                         // Toplam TRIP sayısı
    dwOperationCount: DWORD;                    // Toplam operasyon sayısı
    
    // Son İşlem Bilgisi (SQL buffer)
    stLastOperation: ST_CircuitBreakerOperationRecord;  // SQL'e yazılacak son işlem
    bNewOperationFlag: BOOL;                    // Yeni işlem var, SQL'e yaz
    
    // Arıza İstatistikleri
    dwTotalFaultCount: DWORD;                   // Toplam arıza sayısı
    dwSpringChargeFaultCount: DWORD;            // Yay kurma arıza sayısı
    dwMotionTimeoutCount: DWORD;                // Hareket zaman aşımı sayısı
    dwTripCoilFaultCount: DWORD;                // Trip bobini arıza sayısı
    
    // Bakım Bilgileri
    bMaintenanceRequired: BOOL;                 // Bakım gerekli
    dwRemainingOperations: DWORD;               // Kalan operasyon sayısı
END_STRUCT
END_TYPE

// ---- _ES/13_CircuitBreaker/Structure/ST_CircuitBreakerStatus.TcDUT
TYPE ST_CircuitBreakerStatus :
STRUCT
    ePosition: E_CircuitBreakerPosition;        // Kesici pozisyonu
    eStatus: E_CircuitBreakerStatus;            // Operasyonel durum
    eActiveMode: E_CircuitBreakerControlMode;   // Aktif kontrol modu
    bSpringCharged: BOOL;                       // Yay kurulu durumu
    bFaultActive: BOOL;                         // Arıza durumu
    eFaultCode: E_CircuitBreakerFault;         // Arıza kodu
    bPLCControlActive: BOOL;                    // PLC kontrol durumu
    bOnCommand: BOOL;                           // ON komut çıkışı
    bOffCommand: BOOL;                          // OFF komut çıkışı
    wsStatusText: WSTRING(100);                 // Durum açıklama metni
END_STRUCT
END_TYPE

// ---- _ES/14_CompensationGroup/Enum/E_CompensationError.TcTLEO
// Hata kodları için ENUM
TYPE E_CompensationError :
(
    ERROR_NONE := 0,                        // Hata yok
    ERROR_INVALID_GROUP_COUNT := 1,         // Geçersiz grup sayısı
    ERROR_NEGATIVE_POWER := 2,              // Negatif güç değeri
    ERROR_NEGATIVE_QUANTITY := 3,           // Negatif kondansatör sayısı
    ERROR_MAX_CAPACITOR_EXCEEDED := 4      // Maksimum kondansatör sayısı aşıldı
);
END_TYPE

// ---- _ES/14_CompensationGroup/Structure/ST_CompensationConfigInfo.TcDUT
TYPE ST_CompensationConfigInfo :
STRUCT
    astGroupConfig : ARRAY[0..GVL_CompensationGroup.MAX_COMPENSATION_GROUPS-1] OF ST_CompensationGroup;  // Tüm grup konfigürasyonları
    nConfiguredGroups : INT;                                                                             // Konfigüre edilmiş grup sayısı
END_STRUCT
END_TYPE

// ---- _ES/14_CompensationGroup/Structure/ST_CompensationDiagnostic.TcDUT
TYPE ST_CompensationDiagnostic :
STRUCT
    bError : BOOL;                          // Hata durumu
    eError : E_CompensationError;           // Hata kodu
    wsErrorMessage : WSTRING(255);          // Hata mesajı
END_STRUCT
END_TYPE

// ---- _ES/14_CompensationGroup/Structure/ST_CompensationGroup.TcDUT
// Kondansatör grubu yapısı
TYPE ST_CompensationGroup :
STRUCT
    rPower : REAL;                                                      // Tek kondansatörün gücü (kVAr)
    rVoltage : REAL;                                                    // Kondansatör gerilimi (V)
    nQuantity : INT;                                                    // Gruptaki kondansatör sayısı
    sTagPrefix : STRING(GVL_CompensationGroup.MAX_TAG_LENGTH);         // Kondansatör etiket öneki
    sProductCode : STRING(GVL_CompensationGroup.MAX_PRODUCT_CODE_LENGTH); // Ürün kodu
END_STRUCT
END_TYPE

// ---- _ES/14_CompensationGroup/Structure/ST_CompensationGroupDetails.TcDUT
TYPE ST_CompensationGroupDetails :
STRUCT
    abGroupActive : ARRAY[0..GVL_CompensationGroup.MAX_COMPENSATION_GROUPS-1] OF BOOL;     // Hangi gruplar aktif
    arGroupPower : ARRAY[0..GVL_CompensationGroup.MAX_COMPENSATION_GROUPS-1] OF REAL;      // Her grubun toplam gücü
    anGroupCapacitorCount : ARRAY[0..GVL_CompensationGroup.MAX_COMPENSATION_GROUPS-1] OF INT; // Her gruptaki kondansatör sayısı
END_STRUCT
END_TYPE

// ---- _ES/14_CompensationGroup/Structure/ST_CompensationHMI.TcDUT
TYPE ST_CompensationHMI :
STRUCT
    stSummary : ST_CompensationSummary;            // Özet bilgiler
    stDiagnostic : ST_CompensationDiagnostic;      // Diagnostik bilgiler
    stGroupDetails : ST_CompensationGroupDetails;   // Grup detayları
    stConfig : ST_CompensationConfigInfo;           // Konfigürasyon bilgileri
END_STRUCT
END_TYPE

// ---- _ES/14_CompensationGroup/Structure/ST_CompensationSummary.TcDUT
TYPE ST_CompensationSummary :
STRUCT
    nTotalActiveCapacitors : INT;           // Toplam aktif kondansatör sayısı
    rTotalActivePower : REAL;               // Toplam aktif güç (kVAr)
    nActiveGroupCount : INT;                // Aktif grup sayısı
END_STRUCT
END_TYPE

// ---- _ES/xx_Line/Enum/E_LineColors.TcDUT
TYPE E_LineColors :
(
	Default := 0,
	Energised_Red := 1,
	Grounded_Green := 2,
	Scnerio_SelectionPurple := 3,
	Optional_SelectionOrange :=4,
	Error := 5
);
END_TYPE

// ---- _ES/xx_Line/Structure/ST_CapacitorSchemaColorBase.TcDUT
TYPE ST_CapacitorSchemaColorBase :
STRUCT
	TopLineColor : E_LineColors;
	BottomLineColor : E_LineColors;
	BottomLineColor2 : E_LineColors;
	CapacitorColor : E_LineColors;
	GroundColor : E_LineColors;
END_STRUCT
END_TYPE

// ---- _ES/xx_Line/Structure/ST_CapacitorSchemaColorWithContactor.TcDUT
TYPE ST_CapacitorSchemaColorWithContactor EXTENDS ST_CapacitorSchemaColorBase :
STRUCT
		ContactorPosition : E_ContactorPosition;
END_STRUCT
END_TYPE

// ---- _ES/xx_Line/Structure/ST_CapacitorSchemaColorWithDisconnector.TcDUT
TYPE ST_CapacitorSchemaColorWithDisconnector EXTENDS ST_CapacitorSchemaColorBase :
STRUCT
	DisconnectorPosition : E_DisconnectorPosition;
END_STRUCT
END_TYPE

// ---- POUs/Alarm/GVL_Alarm.TcGVL
{attribute 'qualified_only'}
VAR_GLOBAL
	bMasterReset		: BOOL;
	bSafetyLoop			: BOOL;
	
	EP6_3X2_24VDC_OK	AT %I*	: BOOL;
	EP6_UPS_24VDC_OK	AT %I*	: BOOL;
	
	EP7_3X2_24VDC_OK	AT %I*	: BOOL;
	EP7_UPS_24VDC_OK	AT %I*	: BOOL;	
	
	EP8_3X2_24VDC_OK	AT %I*	: BOOL;
	EP8_UPS_24VDC_OK	AT %I*	: BOOL;		
	
	EP9_3X2_24VDC_OK	AT %I*	: BOOL;
	EP9_UPS_24VDC_OK	AT %I*	: BOOL;		
	
	EP10_3X2_24VDC_OK	AT %I*	: BOOL;
	EP10_UPS_24VDC_OK	AT %I*	: BOOL;		
END_VAR

// ---- POUs/Example/GVL_HMI.TcGVL
VAR_GLOBAL
    // Disconnector 1 HMI verileri
    stDisconnector1_HMI: ST_DisconnectorHMI;
    
    // Contactor 1 HMI verileri
    stContactor1_HMI: ST_ContactorHMI;
	
    // Circuit Breaker 1 HMI verileri
    stCircuitBreaker1_HMI: ST_CircuitBreakerHMI;	
END_VAR

// ---- POUs/Example/GVL_IO.TcGVL
VAR_GLOBAL
    // Disconnector 1 IO Structure
    stDisconnector1_IO: ST_DisconnectorIO;
    
    // Contactor 1 IO Structure  
    stContactor1_IO: ST_ContactorIO;
	
    // IO Structure
    stCircuitBreaker1_IO: ST_CircuitBreakerIO;	
END_VAR

// ---- POUs/Example/GVL_Safety.TcGVL
VAR_GLOBAL
    bSafetyLoop: BOOL;                          // Genel safety loop
    bDisconnector1_Interlock: BOOL;             // Ayırıcı 1 interlock
    bContactor1_Interlock: BOOL;                // Kontaktör 1 interlock
    bCircuitBreaker1_Interlock: BOOL;           // Kesici 1 interlock
END_VAR

// ---- POUs/Example/GVL_System.TcGVL
VAR_GLOBAL
    bMasterReset: BOOL;                               // Sistem master reset
END_VAR

// ---- POUs/HVCP3/GVL_HVCP3.TcGVL
{attribute 'qualified_only'}
VAR_GLOBAL
    // Kompanzasyon grupları konfigürasyonu
    astCompensationGroups : ARRAY[0..GVL_CompensationGroup.MAX_COMPENSATION_GROUPS-1] OF ST_CompensationGroup;  // Tüm grupların kondansatör bilgileri
    nConfiguredGroups : INT;                                                                                    // Toplam konfigüre edilmiş grup sayısı
    
    // Grup aktif durumları
    abGroupActive : ARRAY[0..GVL_CompensationGroup.MAX_COMPENSATION_GROUPS-1] OF BOOL;                         // Her grubun aktif/pasif durumu

    // Ana kesici HMI bilgileri
    stMainDisconnectorHMI : ST_DisconnectorHMI;                                                               // Ana kesici durum ve kontrol bilgileri	
	
	// 12CB1 kesici HMI bilgileri
	st12CB1HMI : ST_DisconnectorHMI;		// 12CB1 kesici durum ve kontrol bilgileri		
	
	// 14CB1 kesici HMI bilgileri
	st14CB1HMI : ST_DisconnectorHMI;		// 14CB1 kesici durum ve kontrol bilgileri	
	
	// 16CB1 kesici HMI bilgileri
	st16CB1HMI : ST_DisconnectorHMI;		// 16CB1 kesici durum ve kontrol bilgileri
	
	// 18CB1 kesici HMI bilgileri
	st18CB1HMI : ST_DisconnectorHMI;		// 18CB1 kesici durum ve kontrol bilgileri
	
	// 20CB1 kesici HMI bilgileri
	st20CB1HMI : ST_DisconnectorHMI;		// 20CB1 kesici durum ve kontrol bilgileri
	
	// 22CB1 kesici HMI bilgileri
	st22CB1HMI : ST_DisconnectorHMI;		// 22CB1 kesici durum ve kontrol bilgileri
	
	// 24CB1 kesici HMI bilgileri
	st24CB1HMI : ST_DisconnectorHMI;		// 24CB1 kesici durum ve kontrol bilgileri
	
	// 26CB1 kesici HMI bilgileri
	st26CB1HMI : ST_DisconnectorHMI;		// 26CB1 kesici durum ve kontrol bilgileri
	
	// 28CB1 kesici HMI bilgileri
	st28CB1HMI : ST_DisconnectorHMI;		// 28CB1 kesici durum ve kontrol bilgileri
	
	// 30CB1 kesici HMI bilgileri
	st30CB1HMI : ST_DisconnectorHMI;		// 30CB1 kesici durum ve kontrol bilgileri
	
	// 32CB1 kesici HMI bilgileri
	st32CB1HMI : ST_DisconnectorHMI;		// 32CB1 kesici durum ve kontrol bilgileri
	
	// 34CB1 kesici HMI bilgileri
	st34CB1HMI : ST_DisconnectorHMI;		// 34CB1 kesici durum ve kontrol bilgileri
	
	// 36CB1 kesici HMI bilgileri
	st36CB1HMI : ST_DisconnectorHMI;		// 36CB1 kesici durum ve kontrol bilgileri
	
	// 38CB1 kesici HMI bilgileri
	st38CB1HMI : ST_DisconnectorHMI;		// 38CB1 kesici durum ve kontrol bilgileri
	
	// 40CB1 kesici HMI bilgileri
	st40CB1HMI : ST_DisconnectorHMI;		// 40CB1 kesici durum ve kontrol bilgileri
	
	// 42CB1 kesici HMI bilgileri
	st42CB1HMI : ST_DisconnectorHMI;		// 42CB1 kesici durum ve kontrol bilgileri
	
	// 44CB1 kesici HMI bilgileri
	st44CB1HMI : ST_DisconnectorHMI;		// 44CB1 kesici durum ve kontrol bilgileri
	
	// 46CB1 kesici HMI bilgileri
	st46CB1HMI : ST_DisconnectorHMI;		// 46CB1 kesici durum ve kontrol bilgileri
	
	// 48CB1 kesici HMI bilgileri
	st48CB1HMI : ST_DisconnectorHMI;		// 48CB1 kesici durum ve kontrol bilgileri
	
	// 50CB1 kesici HMI bilgileri
	st50CB1HMI : ST_DisconnectorHMI;		// 50CB1 kesici durum ve kontrol bilgileri
	
	// 52CB1 kesici HMI bilgileri
	st52CB1HMI : ST_DisconnectorHMI;		// 52CB1 kesici durum ve kontrol bilgileri
	
	// 54CB1 kesici HMI bilgileri
	st54CB1HMI : ST_DisconnectorHMI;		// 54CB1 kesici durum ve kontrol bilgileri
	
	// 56CB1 kesici HMI bilgileri
	st56CB1HMI : ST_DisconnectorHMI;		// 56CB1 kesici durum ve kontrol bilgileri
	
END_VAR

// ---- POUs/HVCP5/GVL_HVCP5.TcGVL
{attribute 'qualified_only'}
VAR_GLOBAL
    // Kompanzasyon grupları konfigürasyonu
    astCompensationGroups : ARRAY[0..GVL_CompensationGroup.MAX_COMPENSATION_GROUPS-1] OF ST_CompensationGroup;  // Tüm grupların kondansatör bilgileri
    nConfiguredGroups : INT;                                                                                    // Toplam konfigüre edilmiş grup sayısı
    
    // Grup aktif durumları
    abGroupActive : ARRAY[0..GVL_CompensationGroup.MAX_COMPENSATION_GROUPS-1] OF BOOL;                         // Her grubun aktif/pasif durumu

    // Ana kesici HMI bilgileri
    st10CB1HMI : ST_DisconnectorHMI;                                                               // Ana kesici durum ve kontrol bilgileri	
	
	// 12CB1 kesici HMI bilgileri
	st12CB1HMI : ST_DisconnectorHMI;		// 12CB1 kesici durum ve kontrol bilgileri		
	
	// 14CB1 kesici HMI bilgileri
	st14CB1HMI : ST_DisconnectorHMI;		// 14CB1 kesici durum ve kontrol bilgileri	
	
	// 16CB1 kesici HMI bilgileri
	st16CB1HMI : ST_DisconnectorHMI;		// 16CB1 kesici durum ve kontrol bilgileri
	
	// 18CB1 kesici HMI bilgileri
	st18CB1HMI : ST_DisconnectorHMI;		// 18CB1 kesici durum ve kontrol bilgileri
	
	// 20CB1 kesici HMI bilgileri
	st20CB1HMI : ST_DisconnectorHMI;		// 20CB1 kesici durum ve kontrol bilgileri
	
	// 22CB1 kesici HMI bilgileri
	st22CB1HMI : ST_DisconnectorHMI;		// 22CB1 kesici durum ve kontrol bilgileri
	
	// 24CB1 kesici HMI bilgileri
	st24CB1HMI : ST_DisconnectorHMI;		// 24CB1 kesici durum ve kontrol bilgileri
	
	// 26CB1 kesici HMI bilgileri
	st26CB1HMI : ST_DisconnectorHMI;		// 26CB1 kesici durum ve kontrol bilgileri
	
	// 28CB1 kesici HMI bilgileri
	st28CB1HMI : ST_DisconnectorHMI;		// 28CB1 kesici durum ve kontrol bilgileri
	
	// 30CB1 kesici HMI bilgileri
	st30CB1HMI : ST_DisconnectorHMI;		// 30CB1 kesici durum ve kontrol bilgileri
	
	// 32CB1 kesici HMI bilgileri
	st32CB1HMI : ST_DisconnectorHMI;		// 32CB1 kesici durum ve kontrol bilgileri
	
	// 34CB1 kesici HMI bilgileri
	st34CB1HMI : ST_DisconnectorHMI;		// 34CB1 kesici durum ve kontrol bilgileri
	
	// 36CB1 kesici HMI bilgileri
	st36CB1HMI : ST_DisconnectorHMI;		// 36CB1 kesici durum ve kontrol bilgileri
	
	// 38CB1 kesici HMI bilgileri
	st38CB1HMI : ST_DisconnectorHMI;		// 38CB1 kesici durum ve kontrol bilgileri

END_VAR

// ---- POUs/LVCP1/GVL_LVCP1.TcGVL
{attribute 'qualified_only'}
VAR_GLOBAL PERSISTENT

    // Kompanzasyon grupları konfigürasyonu
    astCompensationGroups : ARRAY[0..GVL_CompensationGroup.MAX_COMPENSATION_GROUPS-1] OF ST_CompensationGroup;  // Tüm grupların kondansatör bilgileri
    nConfiguredGroups : INT;                                                                                    // Toplam konfigüre edilmiş grup sayısı
    
    // Grup aktif durumları
    abGroupActive : ARRAY[0..GVL_CompensationGroup.MAX_COMPENSATION_GROUPS-1] OF BOOL;                         // Her grubun aktif/pasif durumu
    
    // Ana kesici HMI bilgileri
    stMainDisconnectorHMI : ST_DisconnectorHMI;                                                               // Ana kesici durum ve kontrol bilgileri
    
    // Grup 1 Kontaktör HMI bilgileri
    stGroup1_ContactorHMI : ST_ContactorHMI;                                                                   // Grup 1 kontaktör durum ve kontrol bilgileri
    
    // Grup 2 Kontaktör HMI bilgileri
    stGroup2_ContactorHMI : ST_ContactorHMI;                                                                   // Grup 2 kontaktör durum ve kontrol bilgileri
    
    // Grup 3 Kontaktör HMI bilgileri
    stGroup3_ContactorHMI : ST_ContactorHMI;                                                                   // Grup 3 kontaktör durum ve kontrol bilgileri
    
    // Grup 4 Kontaktör HMI bilgileri
    stGroup4_ContactorHMI : ST_ContactorHMI;                                                                   // Grup 4 kontaktör durum ve kontrol bilgileri
    
    // Grup 5 Kontaktör HMI bilgileri
    stGroup5_ContactorHMI : ST_ContactorHMI;                                                                   // Grup 5 kontaktör durum ve kontrol bilgileri
    
    // Grup 6 Kontaktör HMI bilgileri
    stGroup6_ContactorHMI : ST_ContactorHMI;                                                                   // Grup 6 kontaktör durum ve kontrol bilgileri
   
   // Grup 7 Kontaktör HMI bilgileri
   stGroup7_ContactorHMI : ST_ContactorHMI;                                                                   // Grup 7 kontaktör durum ve kontrol bilgileri
   
   // Grup 8 Kontaktör HMI bilgileri
   stGroup8_ContactorHMI : ST_ContactorHMI;                                                                   // Grup 8 kontaktör durum ve kontrol bilgileri
   
   // Grup 9 Kontaktör HMI bilgileri
   stGroup9_ContactorHMI : ST_ContactorHMI;                                                                   // Grup 9 kontaktör durum ve kontrol bilgileri
   
   // Grup 10 Kontaktör HMI bilgileri
   stGroup10_ContactorHMI : ST_ContactorHMI;                                                                  // Grup 10 kontaktör durum ve kontrol bilgileri
END_VAR

// ---- POUs/LVCP2/GVL_LVCP2.TcGVL
{attribute 'qualified_only'}
VAR_GLOBAL PERSISTENT
	// stPower	
	stEnergyData	: MDP5001_341_EDB8EE3C; 
	
    // Kompanzasyon grupları konfigürasyonu
    astCompensationGroups : ARRAY[0..GVL_CompensationGroup.MAX_COMPENSATION_GROUPS-1] OF ST_CompensationGroup;  // Tüm grupların kondansatör bilgileri
    nConfiguredGroups : INT;                                                                                    // Toplam konfigüre edilmiş grup sayısı
    
    // Grup aktif durumları
    abGroupActive : ARRAY[0..GVL_CompensationGroup.MAX_COMPENSATION_GROUPS-1] OF BOOL;                         // Her grubun aktif/pasif durumu
    
    // Ana kesici HMI bilgileri
    stMainDisconnectorHMI : ST_DisconnectorHMI;                                                               // Ana kesici durum ve kontrol bilgileri
    
    // Grup 1 Kontaktör HMI bilgileri
    stGroup1_ContactorHMI : ST_ContactorHMI;                                                                   // Grup 1 kontaktör durum ve kontrol bilgileri
    
    // Grup 2 Kontaktör HMI bilgileri
    stGroup2_ContactorHMI : ST_ContactorHMI;                                                                   // Grup 2 kontaktör durum ve kontrol bilgileri
    
    // Grup 3 Kontaktör HMI bilgileri
    stGroup3_ContactorHMI : ST_ContactorHMI;                                                                   // Grup 3 kontaktör durum ve kontrol bilgileri
    
    // Grup 4 Kontaktör HMI bilgileri
    stGroup4_ContactorHMI : ST_ContactorHMI;                                                                   // Grup 4 kontaktör durum ve kontrol bilgileri
    
    // Grup 5 Kontaktör HMI bilgileri
    stGroup5_ContactorHMI : ST_ContactorHMI;                                                                   // Grup 5 kontaktör durum ve kontrol bilgileri
    
    // Grup 6 Kontaktör HMI bilgileri
    stGroup6_ContactorHMI : ST_ContactorHMI;                                                                   // Grup 6 kontaktör durum ve kontrol bilgileri
   
   // Grup 7 Kontaktör HMI bilgileri
   stGroup7_ContactorHMI : ST_ContactorHMI;                                                                   // Grup 7 kontaktör durum ve kontrol bilgileri
   
   // Grup 8 Kontaktör HMI bilgileri
   stGroup8_ContactorHMI : ST_ContactorHMI;                                                                   // Grup 8 kontaktör durum ve kontrol bilgileri
   
   // Grup 9 Kontaktör HMI bilgileri
   stGroup9_ContactorHMI : ST_ContactorHMI;                                                                   // Grup 9 kontaktör durum ve kontrol bilgileri
   
   // Grup 10 Kontaktör HMI bilgileri
   stGroup10_ContactorHMI : ST_ContactorHMI;                                                                  // Grup 10 kontaktör durum ve kontrol bilgileri
END_VAR

// ---- POUs/LVCP5/GVL_LVCP5.TcGVL
{attribute 'qualified_only'}
VAR_GLOBAL PERSISTENT
    // Kompanzasyon grupları konfigürasyonu
    astCompensationGroups : ARRAY[0..GVL_CompensationGroup.MAX_COMPENSATION_GROUPS-1] OF ST_CompensationGroup;  // Tüm grupların kondansatör bilgileri
    nConfiguredGroups : INT;                                                                                    // Toplam konfigüre edilmiş grup sayısı
    
    // Grup aktif durumları
    abGroupActive : ARRAY[0..GVL_CompensationGroup.MAX_COMPENSATION_GROUPS-1] OF BOOL;                         // Her grubun aktif/pasif durumu	

    // Ana şalter HMI verileri
    stMainCircuitBreakerHMI: ST_CircuitBreakerHMI;	
	
    // Grup 1 Kontaktör HMI bilgileri
    stGroup1_ContactorHMI : ST_ContactorHMI;                                                                   // Grup 1 kontaktör durum ve kontrol bilgileri
    
    // Grup 2 Kontaktör HMI bilgileri
    stGroup2_ContactorHMI : ST_ContactorHMI;                                                                   // Grup 2 kontaktör durum ve kontrol bilgileri
    
    // Grup 3 Kontaktör HMI bilgileri
    stGroup3_ContactorHMI : ST_ContactorHMI;                                                                   // Grup 3 kontaktör durum ve kontrol bilgileri
    
    // Grup 4 Kontaktör HMI bilgileri
    stGroup4_ContactorHMI : ST_ContactorHMI;                                                                   // Grup 4 kontaktör durum ve kontrol bilgileri
    
    // Grup 5 Kontaktör HMI bilgileri
    stGroup5_ContactorHMI : ST_ContactorHMI;                                                                   // Grup 5 kontaktör durum ve kontrol bilgileri
    
    // Grup 6 Kontaktör HMI bilgileri
    stGroup6_ContactorHMI : ST_ContactorHMI;                                                                   // Grup 6 kontaktör durum ve kontrol bilgileri
   
   // Grup 7 Kontaktör HMI bilgileri
   stGroup7_ContactorHMI : ST_ContactorHMI;	
END_VAR

// ---- _ES/14_CompensationGroup/GVL_CompensationGroup.TcGVL
{attribute 'qualified_only'}
VAR_GLOBAL CONSTANT
    MAX_COMPENSATION_GROUPS : INT := 20;        // Maksimum kompanzasyon grup sayısı
    MAX_TOTAL_CAPACITORS : INT := 100;          // Maksimum toplam kondansatör sayısı
    MAX_TAG_LENGTH : INT := 30;                 // Maksimum etiket uzunluğu
    MAX_PRODUCT_CODE_LENGTH : INT := 50;        // Maksimum ürün kodu uzunluğu
END_VAR

// ---- POUs/MAIN.TcPOU
PROGRAM MAIN
VAR
	lineColor : E_LineColors;
END_VAR

PRG_DisconnectorExample();

PRG_ContactorExample();

PRG_CircuitBreakerExample();

PRG_Simulation();

PRG_LVCP1();

PRG_LVCP2();

PRG_LVCP5();

PRG_HVCP3();

PRG_HVCP5();

END_PROGRAM

// ---- POUs/Example/PRG_DisconnectorExample.TcPOU
PROGRAM PRG_DisconnectorExample
VAR
    // Function Block Instance
    fbDisconnector1: FB_DisconnectorControl;
    
    // Başlangıç konfigürasyonu için flag
    bInitDone: BOOL;
END_VAR


// Function Block Çağrısı
fbDisconnector1(
    // Fiziksel Girişler
    bContactorOn_FB := stDisconnector1_IO.bContactorOn_FB,
    bContactorOff_FB := stDisconnector1_IO.bContactorOff_FB,
    bLimitOn := stDisconnector1_IO.bLimitOn,
    bLimitOff := stDisconnector1_IO.bLimitOff,
    bThermalFault := stDisconnector1_IO.bThermalFault,
    bEarthSwitchOn := stDisconnector1_IO.bEarthSwitchOn,
    bEarthSwitchOff := stDisconnector1_IO.bEarthSwitchOff,
    bPLCControl := stDisconnector1_IO.bPLCControl,
    
    // Güvenlik Girişleri
    bSafetyLoop := GVL_Safety.bSafetyLoop,
    bInterlock := GVL_Safety.bDisconnector1_Interlock,
    
    // Sistem Girişleri
    bMasterReset := GVL_System.bMasterReset,
    
    // HMI Bağlantısı
    stHMI := GVL_HMI.stDisconnector1_HMI,
    
    // Fiziksel Çıkışlar
    bContactorOn_Out => stDisconnector1_IO.bContactorOn_Out,
    bContactorOff_Out => stDisconnector1_IO.bContactorOff_Out
);

END_PROGRAM

// ---- _ES/11_Disconnector/FB_DisconnectorControl.TcPOU
FUNCTION_BLOCK FB_DisconnectorControl
VAR_INPUT
    // Fiziksel Girişler
    bContactorOn_FB: BOOL;                      // ON kontaktörü geri bildirimi
    bContactorOff_FB: BOOL;                     // OFF kontaktörü geri bildirimi
    bLimitOn: BOOL;                             // ON pozisyon limit switch
    bLimitOff: BOOL;                            // OFF pozisyon limit switch
    bThermalFault: BOOL;                        // Motor termik koruma arızası
    bEarthSwitchOn: BOOL;                       // Toprak bıçağı ON pozisyonu
    bEarthSwitchOff: BOOL;                      // Toprak bıçağı OFF pozisyonu
    bPLCControl: BOOL;                          // PLC kontrol seçici
 
	// Güvenlik Girişleri
	bSafetyLoop: BOOL;                          // Safety loop (Emergency stop chain)
   
    // Güvenlik Girişleri
    bInterlock: BOOL;                           // Dış interlock sinyali
    
    // Sistem Girişleri
    bMasterReset: BOOL;                         // Master reset (tüm arıza ve istatistikleri sıfırlar)
END_VAR

VAR_OUTPUT
    // Fiziksel Çıkışlar
    bContactorOn_Out: BOOL;                     // ON kontaktörü sürme
    bContactorOff_Out: BOOL;                    // OFF kontaktörü sürme
END_VAR

VAR_IN_OUT
    stHMI: ST_DisconnectorHMI;                 // HMI için tüm veriler
END_VAR

VAR
    // State Machine
    ePosition				: E_DisconnectorPosition;                // İç durum değişkeni
    ePositionPrevious		: E_DisconnectorPosition;        // Önceki durum
    eEarthSwitchPosition	: E_DisconnectorPosition;     // Toprak bıçağı durumu
 
    // Blokaj değişkenleri
    bBlockOn: BOOL;                             // ON hareketi blokaj
    bBlockOff: BOOL;                            // OFF hareketi blokaj
   
    // Timer'lar
    tonMotionTimeout: TON;                      // Hareket zaman aşımı timer'ı
    tonContactorOn: TON;                        // ON kontaktör gecikme timer'ı
    tonContactorOff: TON;                       // OFF kontaktör gecikme timer'ı
    tonEarthSwitchCheckOn: TON;                 // Toprak bıçağı ON kontrolü timer'ı
    tonEarthSwitchCheckOff: TON;                // Toprak bıçağı OFF kontrolü timer'ı
    
    // Edge Detection
    rtrigOnCmd: R_TRIG;                         // ON komut yükselen kenar
    rtrigOffCmd: R_TRIG;                        // OFF komut yükselen kenar
    rtrigResetFault: R_TRIG;                    // Reset yükselen kenar
    rtrigResetStatistics: R_TRIG;               // İstatistik reset yükselen kenar
    rtrigMasterReset: R_TRIG;                   // Master reset yükselen kenar
    
    // İç Değişkenler
    bOnRequest: BOOL;                           // Dahili ON isteği
    bOffRequest: BOOL;                          // Dahili OFF isteği
    tOperationStartTime: TIME;                  // Operasyon başlangıç zamanı
    tCurrentTime: TIME;                         // Şu anki zaman
END_VAR

// Edge Detection
rtrigOnCmd(CLK := bOnRequest);
rtrigOffCmd(CLK := bOffRequest);
rtrigResetFault(CLK := stHMI.stCommand.bResetFault OR bMasterReset);
rtrigResetStatistics(CLK := stHMI.stCommand.bResetStatistics);
rtrigMasterReset(CLK := bMasterReset);

// Reset İşlemleri
IF rtrigResetFault.Q THEN
    A_ResetFault();
END_IF

IF rtrigResetStatistics.Q OR rtrigMasterReset.Q THEN
    A_ResetStatistics();
END_IF

// Ana kontrol akışı
A_ModeSelection();      // Mod seçimi ve komut belirleme
A_PositionCheck();      // Pozisyon güncelleme
A_FaultCheck();         // Arıza kontrolü
A_Control();            // Çıkış kontrolü
A_UpdateStatus();       // Status güncelleme

// Timer'ları çalıştır (sadece geri bildirim gerekli ise)
IF stHMI.stConfig.bContactorFeedbackRequired THEN
    tonContactorOn(IN := bContactorOn_Out AND NOT bContactorOn_FB, PT := stHMI.stConfig.tContactorDelay);
    tonContactorOff(IN := bContactorOff_Out AND NOT bContactorOff_FB, PT := stHMI.stConfig.tContactorDelay);
END_IF

tonMotionTimeout(IN := stHMI.stStatus.bTurningOn OR stHMI.stStatus.bTurningOff, PT := stHMI.stConfig.tMotionTimeout);

// Toprak bıçağı kontrol timer'ları
IF stHMI.stConfig.bEarthSwitchExists AND stHMI.stConfig.bGrounded THEN
    tonEarthSwitchCheckOn(IN := (stHMI.stStatus.ePosition = E_DisconnectorPosition.ON) AND (eEarthSwitchPosition <> E_DisconnectorPosition.OFF), PT := T#5S);
    tonEarthSwitchCheckOff(IN := (stHMI.stStatus.ePosition = E_DisconnectorPosition.OFF) AND (eEarthSwitchPosition <> E_DisconnectorPosition.ON), PT := T#5S);
END_IF

ACTION A_Control:
// ON hareketi blokaj şartları
bBlockOn := bInterlock OR 
            stHMI.stStatus.bFaultActive OR 
            bLimitOn OR 
            stHMI.stCommand.bStop OR 
            NOT bSafetyLoop;

// OFF hareketi blokaj şartları            
bBlockOff := bInterlock OR 
             stHMI.stStatus.bFaultActive OR 
             bLimitOff OR 
             stHMI.stCommand.bStop OR 
             NOT bSafetyLoop;

// ON kontaktör kontrolü
M_OutputControl(
    Invert      := FALSE, 
    Momentary   := bOnRequest, 
    Set         := FALSE,
    Reset       := bBlockOn,  
    Out         => bContactorOn_Out
);

// OFF kontaktör kontrolü  
M_OutputControl(
    Invert      := FALSE, 
    Momentary   := bOffRequest, 
    Set         := FALSE,
    Reset       := bBlockOff,  
    Out         => bContactorOff_Out
);

// Çıkışları status'e kopyala
stHMI.stStatus.bContactorOn_Out := bContactorOn_Out;
stHMI.stStatus.bContactorOff_Out := bContactorOff_Out;
END_ACTION

ACTION A_FaultCheck:
// Her iki limit aktif
IF bLimitOn AND bLimitOff THEN
    ePosition := E_DisconnectorPosition.FAULT;
    stHMI.stStatus.eFaultCode := E_DisconnectorFault.BOTH_LIMITS;
    stHMI.stStatus.bFaultActive := TRUE;
    stHMI.stStatus.wsStatusText := "ARIZA: Her iki limit switch aktif";
END_IF

// Termik arıza
IF bThermalFault THEN
    ePosition := E_DisconnectorPosition.FAULT;
    stHMI.stStatus.eFaultCode := E_DisconnectorFault.THERMAL;
    stHMI.stStatus.bFaultActive := TRUE;
    stHMI.stStatus.wsStatusText := "ARIZA: Motor termik koruma aktif";
END_IF

// ON kontaktör geri bildirim kontrolü (eğer gerekli ise)
IF stHMI.stConfig.bContactorFeedbackRequired THEN
    tonContactorOn(IN := bContactorOn_Out AND NOT bContactorOn_FB, PT := stHMI.stConfig.tContactorDelay);
    IF tonContactorOn.Q THEN
        ePosition := E_DisconnectorPosition.FAULT;
        stHMI.stStatus.eFaultCode := E_DisconnectorFault.CONTACTOR_ON;
        stHMI.stStatus.bFaultActive := TRUE;
        stHMI.stStatus.wsStatusText := "ARIZA: ON kontaktör geri bildirim hatası";
    END_IF

    // OFF kontaktör geri bildirim kontrolü
    tonContactorOff(IN := bContactorOff_Out AND NOT bContactorOff_FB, PT := stHMI.stConfig.tContactorDelay);
    IF tonContactorOff.Q THEN
        ePosition := E_DisconnectorPosition.FAULT;
        stHMI.stStatus.eFaultCode := E_DisconnectorFault.CONTACTOR_OFF;
        stHMI.stStatus.bFaultActive := TRUE;
        stHMI.stStatus.wsStatusText := "ARIZA: OFF kontaktör geri bildirim hatası";
    END_IF
END_IF

// Hareket zaman aşımı kontrolü
tonMotionTimeout(IN := (ePosition = E_DisconnectorPosition.TURNING_ON) OR (ePosition = E_DisconnectorPosition.TURNING_OFF), PT := stHMI.stConfig.tMotionTimeout);
IF tonMotionTimeout.Q THEN
    ePosition := E_DisconnectorPosition.FAULT;
    stHMI.stStatus.eFaultCode := E_DisconnectorFault.MOTION_TIMEOUT;
    stHMI.stStatus.bFaultActive := TRUE;
    stHMI.stStatus.wsStatusText := "ARIZA: Hareket zaman aşımı";
END_IF

// Toprak bıçağı senkronizasyon kontrolü
IF stHMI.stConfig.bEarthSwitchExists AND stHMI.stConfig.bGrounded THEN
    tonEarthSwitchCheckOn(IN := (ePosition = E_DisconnectorPosition.ON) AND (eEarthSwitchPosition <> E_DisconnectorPosition.OFF), PT := T#5S);
    IF tonEarthSwitchCheckOn.Q THEN
        ePosition := E_DisconnectorPosition.FAULT;
        stHMI.stStatus.eFaultCode := E_DisconnectorFault.EARTH_SWITCH;
        stHMI.stStatus.bFaultActive := TRUE;
        stHMI.stStatus.wsStatusText := "ARIZA: Toprak bıçağı senkronizasyon hatası";
    END_IF
    
    tonEarthSwitchCheckOff(IN := (ePosition = E_DisconnectorPosition.OFF) AND (eEarthSwitchPosition <> E_DisconnectorPosition.ON), PT := T#5S);
    IF tonEarthSwitchCheckOff.Q THEN
        ePosition := E_DisconnectorPosition.FAULT;
        stHMI.stStatus.eFaultCode := E_DisconnectorFault.EARTH_SWITCH;
        stHMI.stStatus.bFaultActive := TRUE;
        stHMI.stStatus.wsStatusText := "ARIZA: Toprak bıçağı senkronizasyon hatası";
    END_IF
END_IF
END_ACTION

ACTION A_ModeSelection:

// PLC kontrolü yoksa mod otomatik olarak REMOTE olur
IF NOT bPLCControl THEN
    stHMI.stStatus.eActiveMode := E_DisconnectorControlMode.REMOTE;
    bOnRequest := FALSE;
    bOffRequest := FALSE;
    stHMI.stCommand.bManualOnCmd := FALSE;
    stHMI.stCommand.bManualOffCmd := FALSE;
    RETURN;
END_IF

// PLC kontrolü varsa komut edilen modu kullan (AUTO veya MANUAL)
// REMOTE modu seçili olsa bile, PLC kontrol varsa AUTO'ya geç
IF stHMI.stCommand.eControlMode = E_DisconnectorControlMode.REMOTE THEN
    stHMI.stStatus.eActiveMode := E_DisconnectorControlMode.AUTO;
ELSE
    stHMI.stStatus.eActiveMode := stHMI.stCommand.eControlMode;
END_IF

// STOP komutu kontrolü - öncelikli
IF stHMI.stCommand.bStop OR stHMI.stStatus.bFaultActive THEN
    bOnRequest := FALSE;
    bOffRequest := FALSE;
    stHMI.stCommand.bManualOnCmd := FALSE;
    stHMI.stCommand.bManualOffCmd := FALSE;	
    RETURN;
END_IF

// Kontrol moduna göre komut seçimi
CASE stHMI.stStatus.eActiveMode OF
    E_DisconnectorControlMode.MANUAL:
        bOnRequest := stHMI.stCommand.bManualOnCmd;
        bOffRequest := stHMI.stCommand.bManualOffCmd;
        
    E_DisconnectorControlMode.AUTO:
        bOnRequest := stHMI.stCommand.bAutoOnCmd;
        bOffRequest := stHMI.stCommand.bAutoOffCmd;
END_CASE

// Çift komut kontrolü
IF bOnRequest AND bOffRequest THEN
    bOnRequest := FALSE;
    bOffRequest := FALSE;
END_IF
END_ACTION

ACTION A_PositionCheck:
// Ayırıcı pozisyon kontrolü
IF bLimitOn AND NOT bLimitOff THEN
    ePosition := E_DisconnectorPosition.ON;
ELSIF bLimitOff AND NOT bLimitOn THEN
    ePosition := E_DisconnectorPosition.OFF;
ELSIF NOT bLimitOn AND NOT bLimitOff THEN
    ePosition := E_DisconnectorPosition.UNDEFINED;
END_IF

// Toprak bıçağı pozisyon kontrolü
IF stHMI.stConfig.bEarthSwitchExists THEN
    IF bEarthSwitchOn AND NOT bEarthSwitchOff THEN
        eEarthSwitchPosition := E_DisconnectorPosition.ON;
    ELSIF bEarthSwitchOff AND NOT bEarthSwitchOn THEN
        eEarthSwitchPosition := E_DisconnectorPosition.OFF;
    ELSIF NOT bEarthSwitchOn AND NOT bEarthSwitchOff THEN
        eEarthSwitchPosition := E_DisconnectorPosition.UNDEFINED;
    END_IF
END_IF
END_ACTION

